# B&R Automation Studio project GAT (part 5)

#### FileOperations.st
```iecst
ACTION FileCopyOperation:

//	(* Export/Import recipes to/from USB *)
//    CASE hmiFile.Status.CopyStep OF
//        FILE_COPY_WAIT: (* Wait for export/import command *)
//            IF (hmiFile.Commands.ExportToUSB = TRUE) THEN
//                (* Check if USB device is available *)
//                IF (brsstrlen(ADR(MpFileManagerUIConnect.DeviceList.DeviceNames[1])) > 0) THEN
//
//                    (* USB is available proceed with export: select all files on the CF and trigger copy command *)
//                    IF (MpFileManagerUIConnect.DeviceList.SelectedIndex <> 0) THEN
//                        MpFileManagerUIConnect.DeviceList.SelectedIndex := 0;
//                        MpFileManagerUIConnect.File.MultiSelect := FALSE;
//                    ELSIF (MpFileManagerUIConnect.Status = mpFILE_UI_STATUS_IDLE) THEN
//
//                        IF NOT MpFileManagerUIConnect.File.MultiSelect THEN
//                            MpFileManagerUIConnect.File.MultiSelect := TRUE;
//                            FOR Index := 0 TO 49 DO
//                                MpFileManagerUIConnect.File.List.Items[Index].IsSelected := TRUE;
//                            END_FOR;
//                        ELSIF (brsstrlen(ADR(MpFileManagerUIConnect.File.List.Items[Index].Name)) = 0) THEN
//                            (* No files to copy, cancel operation *)
//                            hmiFile.Commands.ExportToUSB := FALSE;
//                        ELSE
//                            MpFileManagerUIConnect.File.Copy := TRUE;
//                            hmiFile.Status.CopyStep := FILE_COPY_TO_USB;
//                            hmiFile.Commands.ExportToUSB := FALSE;
//                        END_IF
//
//                    END_IF
//
//                ELSE
//                    (* No USB disk available, cancel operation *)
//                    hmiFile.Commands.ExportToUSB := FALSE;
//                END_IF
//
//            ELSIF hmiFile.Commands.ImportFromUSB THEN
//                (* Check if USB device is available *)
//                IF (brsstrlen(ADR(MpFileManagerUIConnect.DeviceList.DeviceNames[1])) > 0) THEN
//                    (* USB is available proceed with import: select all files on the USB and trigger copy command *)
//
//                    IF (MpFileManagerUIConnect.DeviceList.SelectedIndex <> 1) THEN
//                        MpFileManagerUIConnect.DeviceList.SelectedIndex := 1;
//                        MpFileManagerUIConnect.File.MultiSelect := FALSE;
//                    ELSIF MpFileManagerUIConnect.Status = mpFILE_UI_STATUS_IDLE THEN
//
//                        IF NOT MpFileManagerUIConnect.File.MultiSelect THEN
//                            MpFileManagerUIConnect.File.MultiSelect := TRUE;
//                            FOR Index := 0 TO ((SIZEOF(MpFileManagerUIConnect.File.List.Items)/SIZEOF(MpFileManagerUIConnect.File.List.Items[0])) - 1) DO
//                                MpFileManagerUIConnect.File.List.Items[Index].IsSelected := TRUE;
//                            END_FOR
//                        ELSIF (brsstrlen(ADR(MpFileManagerUIConnect.File.List.Items[Index].Name)) = 0) THEN
//                            (* No files to copy, cancel operation *)
//                            hmiFile.Commands.ImportFromUSB := FALSE;
//                        ELSE
//                            MpFileManagerUIConnect.File.Copy := TRUE;
//                            hmiFile.Status.CopyStep := FILE_COPY_FROM_USB;
//                            hmiFile.Commands.ImportFromUSB := FALSE;
//                        END_IF
//
//                    END_IF
//                ELSE
//                    (* No USB disk available, cancel operation *)
//                    hmiFile.Commands.ImportFromUSB := FALSE;
//                END_IF
//
//            END_IF
//
//        FILE_COPY_TO_USB: (* Navigate to USB device and paste files *)
//            IF (MpFileManagerUIConnect.Status = mpFILE_UI_STATUS_IDLE) THEN
//
//                IF (MpFileManagerUIConnect.DeviceList.SelectedIndex <> 1) THEN
//                    MpFileManagerUIConnect.DeviceList.SelectedIndex := 1;
//                    MpFileManagerUIConnect.File.MultiSelect := FALSE;
//                ELSE
//                    MpFileManagerUIConnect.File.Paste := TRUE;
//                END_IF
//
//            END_IF
//
//            IF MpFileManagerUIConnect.Status = mpFILE_UI_STATUS_PASTE THEN
//                hmiFile.Status.CopyStep := FILE_COPY_BUSY;
//            END_IF;
//
//        FILE_COPY_FROM_USB: (* Navigate to CF device and paste files *)
//            IF (MpFileManagerUIConnect.DeviceList.SelectedIndex <> 0) THEN
//                MpFileManagerUIConnect.DeviceList.SelectedIndex := 0;
//                MpFileManagerUIConnect.File.MultiSelect := FALSE;
//            ELSIF (MpFileManagerUIConnect.Status = mpFILE_UI_STATUS_IDLE) THEN
//                MpFileManagerUIConnect.File.Paste := TRUE;
//            END_IF
//
//            IF (MpFileManagerUIConnect.Status = mpFILE_UI_STATUS_PASTE) THEN
//                hmiFile.Status.CopyStep := FILE_COPY_BUSY;
//            END_IF
//
//        FILE_COPY_BUSY: (* Wait for copying done *)
//            IF (MpFileManagerUIConnect.MessageBox.Type = mpFILE_MSG_CONFIRM_OVERWRITE) OR (MpFileManagerUIConnect.MessageBox.Type = mpFILE_MSG_BUSY) THEN
//                (* TODO: Replace by confirm dialog *)
//                MpFileManagerUIConnect.MessageBox.Confirm := TRUE;
//            ELSIF MpFileManagerUIConnect.Status = mpFILE_UI_STATUS_IDLE THEN
//                hmiFile.Status.CopyStep := FILE_COPY_WAIT;
//            END_IF
//
//    END_CASE

END_ACTION
```

#### FIFOOperations.st - not listed in the package file held
```iecst
ACTION FIFOOperation:

	R_TRIG_CheckStatus(CLK := (MpFileManagerUIConnect.Status = mpFILE_UI_STATUS_CHANGE_DIR) OR
		(MpFileManagerUIConnect.Status = mpFILE_UI_STATUS_CHANGE_DEVICE) OR
		(MpFileManagerUIConnect.Status = mpFILE_UI_STATUS_CREATE));

	IF R_TRIG_CheckStatus.Q OR TON_ScanFolder.Q THEN
		HmiFile.Commands.CheckFolder := TRUE;
	END_IF

	// Autodelete oldest files based on scanning option
    CASE HmiFile.Status.DeleteStep OF

		FILE_DELETE_WAIT:
			// Wait for check the correct device selection
			TON_ScanFolder.IN := (HmiFile.Status.CurrentPage <> 'File_page');
			IF TON_ScanFolder.Q THEN
				TON_ScanFolder.IN := FALSE;
				HmiFile.Status.DeleteStep := FILE_SCAN_FOLDER_WAIT;
			END_IF

		FILE_SCAN_FOLDER_WAIT:
			// Wait for check for old files command
			IF (HmiFile.Commands.CheckFolder = TRUE) AND (MpFileManagerUIConnect.Status = mpFILE_UI_STATUS_IDLE) THEN
				HmiFile.Commands.CheckFolder := FALSE;
				HmiFile.Status.DeleteStep := FILE_SELECT_DEVICE;
				HmiFile.Parameters.OldSortOrder := MpFileManagerUIConnect.File.SortOrder;
			END_IF

		FILE_SELECT_DEVICE:
			// Sort by date so the oldest files are at the end
            IF (HmiFile.Status.DeviceName <> HmiFile.Parameters.Fifo.DeviceName) THEN
				FOR i := 0 TO ((SIZEOF(MpFileManagerUIConnect.DeviceList.DeviceNames)/SIZEOF(MpFileManagerUIConnect.DeviceList.DeviceNames[0])) - 1) DO
        			IF HmiFile.Parameters.Fifo.DeviceName = MpFileManagerUIConnect.DeviceList.DeviceNames[i] THEN
						MpFileManagerUIConnect.DeviceList.SelectedIndex := i;
					END_IF
    			END_FOR
            END_IF

            IF (HmiFile.Status.DeviceName = HmiFile.Parameters.Fifo.DeviceName) AND (MpFileManagerUIConnect.Status = mpFILE_UI_STATUS_IDLE) THEN
                HmiFile.Status.DeleteStep := FILE_SORT_BY_DATE;
            END_IF

		FILE_SORT_BY_DATE:
			// Sort by date so the oldest files are at the end
            IF (MpFileManagerUIConnect.File.SortOrder <> mpFILE_SORT_BY_MOD_TIME_DESC) THEN
                MpFileManagerUIConnect.File.SortOrder := mpFILE_SORT_BY_MOD_TIME_DESC;
            ELSIF (MpFileManagerUIConnect.Status = mpFILE_UI_STATUS_IDLE) THEN
                MpFileManagerUIConnect.File.Refresh := TRUE;
            END_IF

            IF (MpFileManagerUIConnect.Status = mpFILE_UI_STATUS_REFRESH) THEN
                HmiFile.Status.DeleteStep := FILE_CHECK_FOR_FILTER;
            END_IF

		FILE_CHECK_FOR_FILTER:
			// Check which delete filter is active
            IF (HmiFile.Parameters.Fifo.FifoType = FILE_FIFO_NUM_OF_FILES) THEN
                HmiFile.Status.DeleteStep := FILE_SELECT_OLDEST_FILES_0;
            ELSIF (HmiFile.Parameters.Fifo.FifoType = FILE_FIFO_SIZE_OF_FOLDER) THEN
				HmiFile.Status.DeleteStep := FILE_CALC_FOLDER_SIZE;
//			ELSIF (HmiFile.Parameters.Fifo.FifoType = FILE_FIFO_OLDER_THAN) THEN
//                HmiFile.Status.DeleteStep := FILE_SORT_BY_DATE;
			END_IF

		FILE_SELECT_OLDEST_FILES_0:
			// Scan and select all file over the filter setting
			IF (MpFileManagerUIConnect.Status = mpFILE_UI_STATUS_IDLE) THEN
				IF MpFileManagerUIConnect.File.PathInfo.FileCount > 1 THEN
           			MpFileManagerUIConnect.File.MultiSelect := TRUE;
				END_IF
				HmiFile.Status.AutoDeleteSelected := 0;
				FOR i := 0 TO ((SIZEOF(HmiFile.Status.FileNames)/SIZEOF(HmiFile.Status.FileNames[0])) - 1) DO
					IF i >= HmiFile.Parameters.Fifo.MaxNumberOfFiles THEN
						MpFileManagerUIConnect.File.List.Items[0].IsSelected := FALSE;
						IF (MpFileManagerUIConnect.File.List.Items[i].ItemType <> mpFILE_ITEM_TYPE_NONE) AND NOT MpFileManagerUIConnect.File.List.Items[i].IsFolder THEN
							MpFileManagerUIConnect.File.List.Items[i].IsSelected := TRUE;
							HmiFile.Status.AutoDeleteSelected := HmiFile.Status.AutoDeleteSelected + 1;
						END_IF
					END_IF
				END_FOR

				IF (HmiFile.Status.AutoDeleteSelected > 0) THEN
					HmiFile.Status.DeleteStep := FILE_DELETE_FILES;
				ELSE
					MpFileManagerUIConnect.File.MultiSelect := FALSE;
					HmiFile.Status.DeleteStep := FILE_RESET_SORT_BY;
				END_IF
			END_IF

		FILE_CALC_FOLDER_SIZE:
			// Calculate the overall file size in the open folder
				HmiFile.Status.FolderSize := 0;
				FOR i := 0 TO ((SIZEOF(HmiFile.Status.FileNames)/SIZEOF(HmiFile.Status.FileNames[0])) - 1) DO
					IF MpFileManagerUIConnect.File.List.Items[i].ItemType <> mpFILE_ITEM_TYPE_FOLDER THEN
						HmiFile.Status.FolderSize := HmiFile.Status.FolderSize + UDINT_TO_REAL(MpFileManagerUIConnect.File.List.Items[i].Size);
					END_IF
				END_FOR
				IF (HmiFile.Status.FolderSize > HmiFile.Parameters.Fifo.MaxFolderSize) THEN
					HmiFile.Status.DeleteStep := FILE_SELECT_OLDEST_FILES_1;
				ELSE
					HmiFile.Status.DeleteStep := FILE_RESET_SORT_BY;
				END_IF

		FILE_SELECT_OLDEST_FILES_1:
			// Scan and select all file over the filter setting
			IF (MpFileManagerUIConnect.Status = mpFILE_UI_STATUS_IDLE) THEN
				MpFileManagerUIConnect.File.List.Items[(MpFileManagerUIConnect.File.PathInfo.FileCount - 1)].IsSelected := TRUE;
				HmiFile.Status.DeleteStep := FILE_DELETE_FILES;
			END_IF

		FILE_DELETE_FILES:
			// Set command to delete the selected oldest files
			IF  (MpFileManagerUIConnect.Status = mpFILE_UI_STATUS_IDLE) THEN
				MpFileManagerUIConnect.File.Delete := TRUE;
			END_IF

			IF (MpFileManagerUIConnect.Status = mpFILE_UI_STATUS_DELETE) THEN
				HmiFile.Status.DeleteStep := FILE_CONFIRM_DELETE;
            END_IF

		FILE_CONFIRM_DELETE:
			// Confirm the file delete
            IF (MpFileManagerUIConnect.MessageBox.Type = mpFILE_MSG_CONFIRM_DELETE) THEN
                MpFileManagerUIConnect.MessageBox.Confirm := TRUE;
            ELSIF (MpFileManagerUIConnect.Status = mpFILE_UI_STATUS_IDLE) AND (MpFileManagerUIConnect.MessageBox.LayerStatus = 1) THEN
				IF (HmiFile.Parameters.Fifo.FifoType = FILE_FIFO_SIZE_OF_FOLDER) THEN
                	HmiFile.Status.DeleteStep := FILE_CALC_FOLDER_SIZE;
				ELSE
					HmiFile.Status.DeleteStep := FILE_RESET_SORT_BY;
					MpFileManagerUIConnect.File.MultiSelect := FALSE;
				END_IF
            END_IF

		FILE_RESET_SORT_BY:
			// Restore old sort order
            IF (MpFileManagerUIConnect.File.SortOrder <> HmiFile.Parameters.OldSortOrder) THEN
                MpFileManagerUIConnect.File.SortOrder := HmiFile.Parameters.OldSortOrder;
            ELSIF (MpFileManagerUIConnect.Status = mpFILE_UI_STATUS_IDLE) THEN
                MpFileManagerUIConnect.File.Refresh := TRUE;
            END_IF

            IF (MpFileManagerUIConnect.Status = mpFILE_UI_STATUS_REFRESH) THEN
                HmiFile.Status.DeleteStep := FILE_DELETE_WAIT;
				IF (MpFileManagerUIConnect.MessageBox.Type = mpFILE_MSG_BUSY) THEN
					MpFileManagerUIConnect.MessageBox.Confirm := TRUE;
				END_IF
            END_IF
	END_CASE

	TON_ScanFolder(PT := DINT_TO_TIME(HmiFile.Parameters.Fifo.ScanInterval * 60000));

END_ACTION
```

### Package Logical/Infrastructure/Usb - Package for USB handling for mapp Framework

### Program Logical/Infrastructure/Usb/UsbMgr (IEC) - Usb manager

#### UsbMgr.st - Init, cyclic, exit code
```iecst
//*********************************************************************************
// Copyright: B&R Industrial Automation GmbH
// Author: B&R Industrial Automation GmbH
// Created: April 12, 2022
// Description: This task automatically detects and (un)links USB storage devices
//*********************************************************************************

PROGRAM _INIT

	DevLinkCtrl.FUB.DevLink_0.enable := FALSE;
	DevLinkCtrl.FUB.DevUnlink_0.enable := FALSE;
	DevLinkCtrl.FUB.UsbNodeGet_0.enable := FALSE;
	DevLinkCtrl.FUB.UsbNodeListGet_0.enable := FALSE;
	DevLinkCtrl.FUB.DevLink_0();
	DevLinkCtrl.FUB.DevUnlink_0();
	DevLinkCtrl.FUB.UsbNodeGet_0();
	DevLinkCtrl.FUB.UsbNodeListGet_0();

	FOR i := 0 TO MAX_IDX_USB_DEV_LIST DO
		AttachedUSB[i] := FALSE;
		gUSBAvailable[i] := FALSE;
	END_FOR

END_PROGRAM

PROGRAM _CYCLIC

	CASE DevLinkCtrl.Step OF
		STATE_WAIT:
			// Update USB info list if the node list has changed
			IF (brsmemcmp(ADR(DevLinkCtrl.Parameters.NodeList), ADR(LastNodeList), SIZEOF(LastNodeList)) <> 0) THEN
				DevLinkCtrl.Commands.GetUSBInfo := TRUE;
				// Preserve the previously created drive information in case the order has changed when unplugging a device
				FOR DevLinkCtrl.Parameters.Index := 0 TO MAX_IDX_USB_DEV_LIST DO
					FOR i := 0 TO MAX_IDX_USB_DEV_LIST DO
						IF ((DevLinkCtrl.Parameters.NodeList[DevLinkCtrl.Parameters.Index] = LastNodeList[i]) AND
							(DevLinkCtrl.Parameters.Index <> i) AND (LastNodeList[i] <> 0)) THEN
							brsmemcpy(ADR(TempUSBInfo), ADR(DevLinkCtrl.Parameters.NodeInfoList[DevLinkCtrl.Parameters.Index]), SIZEOF(TempUSBInfo));
							brsmemcpy(ADR(DevLinkCtrl.Parameters.NodeInfoList[DevLinkCtrl.Parameters.Index]), ADR(DevLinkCtrl.Parameters.NodeInfoList[i]), SIZEOF(TempUSBInfo));
							brsmemcpy(ADR(DevLinkCtrl.Parameters.NodeInfoList[i]), ADR(TempUSBInfo), SIZEOF(TempUSBInfo));
							brsmemcpy(ADR(TempFileDeviceName), ADR(DevLinkCtrl.Parameters.FileDevName[DevLinkCtrl.Parameters.Index]), SIZEOF(TempFileDeviceName));
							brsmemcpy(ADR(DevLinkCtrl.Parameters.FileDevName[DevLinkCtrl.Parameters.Index]), ADR(DevLinkCtrl.Parameters.FileDevName[i]), SIZEOF(TempFileDeviceName));
							brsmemcpy(ADR(DevLinkCtrl.Parameters.FileDevName[i]), ADR(TempFileDeviceName), SIZEOF(TempFileDeviceName));
							TempFileDeviceHandle := DevLinkCtrl.Parameters.FileDevHandle[DevLinkCtrl.Parameters.Index];
							DevLinkCtrl.Parameters.FileDevHandle[DevLinkCtrl.Parameters.Index] := DevLinkCtrl.Parameters.FileDevHandle[i];
							DevLinkCtrl.Parameters.FileDevHandle[i] := TempFileDeviceHandle;
						END_IF
					END_FOR
				END_FOR
				brsmemcpy(ADR(LastNodeList), ADR(DevLinkCtrl.Parameters.NodeList), SIZEOF(LastNodeList));
			END_IF

			FOR DevLinkCtrl.Parameters.Index := 0 TO MAX_IDX_USB_DEV_LIST DO
				// Skip if loading USB list information
				IF DevLinkCtrl.Commands.GetUSBInfo THEN
					EXIT;
				END_IF
				// Always keep devices linked when available
				IF ((DevLinkCtrl.Parameters.FileDevHandle[DevLinkCtrl.Parameters.Index] = 0) AND AttachedUSB[DevLinkCtrl.Parameters.Index]
					AND (DevLinkCtrl.Parameters.NodeList[DevLinkCtrl.Parameters.Index] <> 0)) THEN
					DevLinkCtrl.Commands.DevLink := TRUE;
					EXIT;
				END_IF
				// Unlink device if it is not connected anymore
				IF ((DevLinkCtrl.Parameters.FileDevHandle[DevLinkCtrl.Parameters.Index] <> 0) AND
					(DevLinkCtrl.Parameters.NodeInfoList[DevLinkCtrl.Parameters.Index].interfaceClass <> 8)) THEN
					DevLinkCtrl.Commands.DevUnlink := TRUE;
					EXIT;
				END_IF
			END_FOR

			// Check for USB devices every 3 seconds
			TON_0.PT := t#3s;
			IF (TON_0.Q AND NOT DevLinkCtrl.Commands.GetUSBInfo AND NOT DevLinkCtrl.Commands.DevLink AND NOT DevLinkCtrl.Commands.DevUnlink) THEN
				DevLinkCtrl.Commands.GetUSBList := TRUE;
				TON_0.IN := FALSE;
			ELSE
				TON_0.IN := TRUE;
			END_IF
			TON_0();

			IF DevLinkCtrl.Commands.GetUSBInfo THEN
				// Get USB info Commands
				DevLinkCtrl.Commands.GetUSBInfo := FALSE;
				brsmemset(ADR(DevLinkCtrl.Parameters.NodeInfoList), 0, SIZEOF(DevLinkCtrl.Parameters.NodeInfoList));
				DevLinkCtrl.Step := STATE_GET_USB_INFO;
				DevLinkCtrl.Parameters.Index := 0;
			ELSIF DevLinkCtrl.Commands.GetUSBList THEN
				// Get USB list Commands
				DevLinkCtrl.Commands.GetUSBList := FALSE;
				brsmemset(ADR(DevLinkCtrl.Parameters.NodeList), 0, SIZEOF(DevLinkCtrl.Parameters.NodeList));
				DevLinkCtrl.Step := STATE_GET_USB_LIST;
			ELSIF DevLinkCtrl.Commands.DevLink THEN
				// Link Commands
				DevLinkCtrl.Commands.DevLink := FALSE;
				DevLinkCtrl.Step := STATE_DEV_LINK;
			ELSIF DevLinkCtrl.Commands.DevUnlink THEN
				// Unlink Commands
				DevLinkCtrl.Commands.DevUnlink := FALSE;
				DevLinkCtrl.Step := STATE_DEV_UNLINK;
			END_IF

		STATE_GET_USB_LIST:
			// Set FUB parameters
			DevLinkCtrl.FUB.UsbNodeListGet_0.enable := TRUE;
			DevLinkCtrl.FUB.UsbNodeListGet_0.bufferSize := SIZEOF(DevLinkCtrl.Parameters.NodeList);
			DevLinkCtrl.FUB.UsbNodeListGet_0.pBuffer := ADR(DevLinkCtrl.Parameters.NodeList);

			// Error handling
			IF ((DevLinkCtrl.FUB.UsbNodeListGet_0.status = ERR_OK) OR (DevLinkCtrl.FUB.UsbNodeListGet_0.status = asusbERR_USB_NOTFOUND)) THEN
				DevLinkCtrl.Step := STATE_WAIT;
				DevLinkCtrl.FUB.UsbNodeListGet_0.enable := FALSE;
			ELSIF ((DevLinkCtrl.FUB.UsbNodeListGet_0.status <> ERR_FUB_BUSY) AND (DevLinkCtrl.FUB.UsbNodeListGet_0.status <> ERR_FUB_ENABLE_FALSE)
				AND (DevLinkCtrl.FUB.UsbNodeListGet_0.status <> asusbERR_USB_NOTFOUND)) THEN
				DevLinkCtrl.Step := STATE_ERROR_USB;
				DevLinkCtrl.Parameters.ErrorID := DevLinkCtrl.FUB.UsbNodeListGet_0.status;
				DevLinkCtrl.FUB.UsbNodeListGet_0.enable := FALSE;
			END_IF

			DevLinkCtrl.FUB.UsbNodeListGet_0();

		STATE_GET_USB_INFO:
			// Set FUB parameters
			DevLinkCtrl.FUB.UsbNodeGet_0.bufferSize := SIZEOF(DevLinkCtrl.Parameters.NodeInfoList[DevLinkCtrl.Parameters.Index]);
			DevLinkCtrl.FUB.UsbNodeGet_0.enable := TRUE;
			DevLinkCtrl.FUB.UsbNodeGet_0.nodeId := DevLinkCtrl.Parameters.NodeList[DevLinkCtrl.Parameters.Index];
			DevLinkCtrl.FUB.UsbNodeGet_0.pBuffer := ADR(DevLinkCtrl.Parameters.NodeInfoList[DevLinkCtrl.Parameters.Index]);

			// Check if DevLinkCtrl.Parameters.Index contains an entry
			IF (DevLinkCtrl.Parameters.NodeList[DevLinkCtrl.Parameters.Index] = 0) THEN
				DevLinkCtrl.FUB.UsbNodeGet_0.enable := TRUE;
				brsmemset(ADR(DevLinkCtrl.Parameters.NodeInfoList[DevLinkCtrl.Parameters.Index]), 0, SIZEOF(DevLinkCtrl.Parameters.NodeInfoList[DevLinkCtrl.Parameters.Index]));
				DevLinkCtrl.Parameters.Index := DevLinkCtrl.Parameters.Index + 1;
			END_IF

			// Error handling
			IF (DevLinkCtrl.FUB.UsbNodeGet_0.status = ERR_OK) THEN
				DevLinkCtrl.FUB.UsbNodeGet_0.enable := FALSE;
				DevLinkCtrl.Parameters.Index := DevLinkCtrl.Parameters.Index + 1;
			ELSIF ((DevLinkCtrl.FUB.UsbNodeGet_0.status <> ERR_FUB_BUSY) AND (DevLinkCtrl.FUB.UsbNodeGet_0.status <> ERR_FUB_ENABLE_FALSE)) THEN
				DevLinkCtrl.Step := STATE_ERROR_USB;
				DevLinkCtrl.Parameters.ErrorID := DevLinkCtrl.FUB.UsbNodeGet_0.status;
				DevLinkCtrl.FUB.UsbNodeGet_0.enable := FALSE;
			END_IF

			// End of list reached
			IF (DevLinkCtrl.Parameters.Index > MAX_IDX_USB_DEV_LIST) THEN
				DevLinkCtrl.FUB.UsbNodeGet_0.enable := FALSE;
				DevLinkCtrl.Step := STATE_WAIT;
				FOR DevLinkCtrl.Parameters.Index := 0 TO MAX_IDX_USB_DEV_LIST DO
					IF (DevLinkCtrl.Parameters.NodeInfoList[DevLinkCtrl.Parameters.Index].interfaceClass = 8) THEN
						AttachedUSB[DevLinkCtrl.Parameters.Index] := TRUE;
					ELSE
						AttachedUSB[DevLinkCtrl.Parameters.Index] := FALSE;
						gUSBAvailable[DevLinkCtrl.Parameters.Index] := FALSE;
					END_IF
				END_FOR
			END_IF

			DevLinkCtrl.FUB.UsbNodeGet_0();

		STATE_DEV_LINK:
            // Set FUB parameters
			DevLinkCtrl.FUB.DevLink_0.enable := TRUE;
			DevLinkCtrl.FUB.DevLink_0.pDevice := ADR(DevLinkCtrl.Parameters.FileDevName[DevLinkCtrl.Parameters.Index]);
			DevLinkCtrl.Parameters.LinkParam := '/DEVICE=';
			brsstrcat(ADR(DevLinkCtrl.Parameters.LinkParam), ADR(DevLinkCtrl.Parameters.NodeInfoList[DevLinkCtrl.Parameters.Index].ifName));
			DevLinkCtrl.FUB.DevLink_0.pParam := ADR(DevLinkCtrl.Parameters.LinkParam);

			// Error handling
			IF (DevLinkCtrl.FUB.DevLink_0.status = ERR_OK) THEN
				DevLinkCtrl.Parameters.FileDevHandle[DevLinkCtrl.Parameters.Index] := DevLinkCtrl.FUB.DevLink_0.handle;
				DevLinkCtrl.Step := STATE_WAIT;
				DevLinkCtrl.FUB.DevLink_0.enable := FALSE;
				FOR i := 0 TO MAX_IDX_USB_DEV_LIST DO
					gUSBAvailable[i] := AttachedUSB[i];
				END_FOR
			ELSIF ((DevLinkCtrl.FUB.DevLink_0.status <> ERR_FUB_BUSY) AND (DevLinkCtrl.FUB.DevLink_0.status <> ERR_FUB_ENABLE_FALSE)) THEN
				DevLinkCtrl.Step := STATE_ERROR_USB;
				DevLinkCtrl.Parameters.ErrorID := DevLinkCtrl.FUB.DevLink_0.status;
				DevLinkCtrl.FUB.DevLink_0.enable := FALSE;
			END_IF

			DevLinkCtrl.FUB.DevLink_0();

		STATE_DEV_UNLINK:
			// Set FUB parameters
			DevLinkCtrl.FUB.DevUnlink_0.enable := TRUE;
			DevLinkCtrl.FUB.DevUnlink_0.handle := DevLinkCtrl.Parameters.FileDevHandle[DevLinkCtrl.Parameters.Index];

			// Check if we have a handle
			IF (DevLinkCtrl.Parameters.FileDevHandle[DevLinkCtrl.Parameters.Index] = 0) THEN
				DevLinkCtrl.FUB.DevUnlink_0.enable := FALSE;
				DevLinkCtrl.Step := STATE_WAIT;
			END_IF

			// Error handling
			IF (DevLinkCtrl.FUB.DevUnlink_0.status = ERR_OK) THEN
				DevLinkCtrl.Parameters.FileDevHandle[DevLinkCtrl.Parameters.Index] := 0;
				DevLinkCtrl.FUB.DevUnlink_0.enable := FALSE;
				DevLinkCtrl.Step := STATE_WAIT;
			ELSIF ((DevLinkCtrl.FUB.DevUnlink_0.status <> ERR_FUB_BUSY) AND (DevLinkCtrl.FUB.DevUnlink_0.status <> ERR_FUB_ENABLE_FALSE)) THEN
				DevLinkCtrl.Step := STATE_ERROR_USB;
				DevLinkCtrl.Parameters.ErrorID := DevLinkCtrl.FUB.DevUnlink_0.status;
				DevLinkCtrl.FUB.DevUnlink_0.enable := FALSE;
			END_IF

			DevLinkCtrl.FUB.DevUnlink_0();

		STATE_ERROR_USB:
			// Delete error ID and go back to wait step when error is acknowledged
			IF DevLinkCtrl.Commands.ErrAck THEN
				DevLinkCtrl.Parameters.ErrorID := 0;
				DevLinkCtrl.Commands.ErrAck := FALSE;
				DevLinkCtrl.Step := STATE_WAIT;
			END_IF

	END_CASE;

END_PROGRAM

PROGRAM _EXIT

	// Insert code here

END_PROGRAM
```

#### UsbMgr.typ - Local data types
```iecst
(*********************************************************************************
 * Copyright: Bernecker + Rainer
 * Author:    MITC
 * Created:   21 October, 2015/1:30 PM
 *********************************************************************************
 * DevLinkTask data types of project
 *********************************************************************************)

TYPE
	StepType :
		( (*enumeration of the possible machine states*)
		STATE_WAIT := 0, (*waiting for cmds*)
		STATE_GET_USB_LIST, (*getting list of usb devices*)
		STATE_GET_USB_INFO, (*getting info from a usb device*)
		STATE_DEV_LINK, (*linking device*)
		STATE_DEV_UNLINK, (*unlinking device*)
		STATE_ERROR_USB (*some FUB returned an error*)
		);
	CommandType : 	STRUCT  (*possible machine cmds*)
		GetUSBList : BOOL; (*get usb list cmd*)
		GetUSBInfo : BOOL; (*get usb info cmd*)
		DevLink : BOOL; (*link cmd*)
		DevUnlink : BOOL; (*unlink cmd*)
		ErrAck : BOOL; (*error acknowledge cmd*)
	END_STRUCT;
	DevLink_FUBType : 	STRUCT  (*contains all needed FileIO FUBs*)
		UsbNodeListGet_0 : UsbNodeListGet;
		UsbNodeGet_0 : UsbNodeGet;
		UsbMsDeviceReady_0 : UsbMsDeviceReady;
		DevLink_0 : DevLink;
		DevUnlink_0 : DevUnlink;
	END_STRUCT;
	DevLinkCtrlType : 	STRUCT  (*Control structure which contains everything necessary for the file handling machine*)
		Step : StepType; (*actual step*)
		Cmd : CommandType; (*when in STATE_WAIT a cmd with value true will change the machine state*)
		FUB : DevLink_FUBType; (*all DevLink FUBs*)
		Params : ParamsType; (*parameters like file device, error ID, Buffer, ...*)
	END_STRUCT;
	ParamsType : 	STRUCT  (*Parameter structure*)
		ErrorID : UINT; (*the error id from a FUB is stored here in case of error*)
		NodeList : ARRAY[0..MAX_IDX_USB_DEV_LIST]OF UDINT; (*List of connected usb devices*)
		NodeInfoList : ARRAY[0..MAX_IDX_USB_DEV_LIST]OF usbNode_typ; (*Buffer for usb info*)
		FileDevName : ARRAY[0..MAX_IDX_USB_DEV_LIST]OF STRING[30]; (*file device names*)
		FileDevHandle : ARRAY[0..MAX_IDX_USB_DEV_LIST]OF UDINT; (*needed for unlinking the device again*)
		LinkParam : STRING[30]; (*param string to link a device*)
		Index : USINT; (*list index*)
	END_STRUCT;
END_TYPE
```

#### UsbMgr.var - Local variables
```iecst
(*Function Blocks*)
VAR
	TON_0 : TON; (*Tiimer to refresh available usb devices*)
END_VAR
(*Structure Types*)
VAR
	DevLinkCtrl : DevLinkControlType := (0); (*DevLink control structure*)
	TempUSBInfo : usbNode_typ := (0); (*Temporary info structure*)
END_VAR
(*Variables*)
VAR
	LastNodeList : ARRAY[0..MAX_IDX_USB_DEV_LIST] OF UDINT; (*Temporary variable to check if the node list has changed*)
	AttachedUSB : ARRAY[0..MAX_IDX_USB_DEV_LIST] OF BOOL := [2(FALSE)]; (*Flags for whether the USB devices are detected*)
	TempFileDeviceName : STRING[30] := ''; (*Temporary file device name*)
	TempFileDeviceHandle : UDINT := 0; (*Temporary file device handle*)
	i : USINT := 0; (*index to loop through ussb devices*)
	tempDigit : STRING[80];
END_VAR
```

### Package Logical/Infrastructure/Report - Package for mapp Report Framework

### Program Logical/Infrastructure/Report/ReportMgr (IEC) - Report manager

#### ReportMgt.var
```iecst
(********************************************************************
 * COPYRIGHT -- Bernecker + Rainer
 ********************************************************************
 * Program: FolderHandling
 * File: FolderHandling.var
 * Author: Bernecker + Rainer
 * Created: December , 2020
 ********************************************************************
 * Local variables of program Alarm Management
 ********************************************************************)
(*Function Block Declaration*)
VAR
	MpFileManagerUIConnect : MpFileManagerUIConnectType := (DeviceList:=(DeviceNames:=['mappReportFiles',9('')]));
	MpFileManagerUI_0 : MpFileManagerUI;
	TON_0 : TON := (0); (*Timer to wait before refresh*)
	MpReportCore_0 : MpReportCore := (0); (*Core variable for MpReport*)
	LanguageSelect_0 : LanguageSelect := (LanguageSelection:=['en','de'],SelectedIndex:=0);
	DirCreate_0 : DirCreate;
END_VAR
(*Report Management Variables*)
VAR
	EnableDelete : BOOL := TRUE; (*HMI control bit*)
	EnableGenerate : BOOL := TRUE; (*HMI control bit*)
	Refresh : BOOL := 0; (*strrt refresh process*)
	StartGenerate : BOOL := 0; (*variable for interaction with Visualization*)
	DeleteReport : BOOL := 0; (*Start deleting a Report*)
	i : USINT := 0; (*index for save filenames in a array*)
	DisplayFileNameIndex : USINT := 0; (*index of selected file for display in table in mappView*)
	DisplayFileName : ARRAY[0..49] OF STRING[255] := [50('')]; (*Displayed Files for mappView*)
	SetLanguage : STRING[80] := ''; (*Set the current language*)
	TableConfig : STRING[80];
	StrSelectedFile : STRING[256] := '0'; (*Gives the path of selected report to pdfViewer in mappView*)
END_VAR
(*Constants*)
VAR CONSTANT
	REPORT_DEVICE : STRING[80] := 'mappReportFiles'; (*Constant contains filedevice for save reports *)
	REPORT_NAME : STRING[80] := 'Report'; (*Constant contains name of Report*)
	STR_FILE_DEVICE : STRING[80] := '/FileDevice:mappReport/'; (*File Device*)
	LOCAL_FOLDER : STRING[10] := 'Report';
END_VAR
```

#### ReportMgt.st
```iecst
//*********************************************************************************
//* Copyright: B&R Industrial Automation GmbH
//* Author:    B&R Industrial Automation GmbH
//* Created:   30. Sep 2020/08:00
//* Description: Tasks FOR report control. The Report Control handling is done in this task.
//********************************************************************************

PROGRAM _INIT

	// Create folder for this component on the user file device
	DirCreate_0(enable := TRUE, pDevice := ADR('UserPartition'), pName := ADR(LOCAL_FOLDER));

	// Check if folder already exist and if so disabled the function block call
	IF DirCreate_0.status = fiERR_DIR_ALREADY_EXIST THEN
		DirCreate_0(enable := FALSE);
	END_IF

	// Init mapp function blocks
	MpReportCore_0.Enable := TRUE;
	MpReportCore_0.MpLink := ADR(gMpLinkReport);
	MpReportCore_0.Name := ADR(REPORT_NAME);
	MpReportCore_0.DeviceName := ADR(REPORT_DEVICE);
	MpFileManagerUI_0.MpLink := ADR(gMpLinkFileManagerUIReport);
	MpFileManagerUI_0.UIConnect := ADR(MpFileManagerUIConnect);
	MpFileManagerUI_0.Enable := TRUE;
	// Filter for pdf files
	MpFileManagerUIConnect.File.Filter := '*.pdf';
END_PROGRAM

PROGRAM _CYCLIC
	// Configure visible file list
	brsstrcpy(ADR(TableConfig), ADR('{ "specRows": [{"from":'));
	brsitoa(MpFileManagerUIConnect.File.PathInfo.FileCount, ADR(TableConfig) + brsstrlen(ADR(TableConfig)));
	brsstrcat(ADR(TableConfig),  ADR(',"to":49, "visible":false}]}'));

	// Refresh report action
	RefreshReport;

	// Reset ErrorReset command
	IF NOT MpReportCore_0.Error THEN
		MpReportCore_0.ErrorReset := FALSE;
	END_IF

	// Function block calls
	MpReportCore_0();
	MpFileManagerUI_0();
END_PROGRAM

PROGRAM _EXIT
	// Disable and call mapp function blocks
	MpReportCore_0.Enable := FALSE;
	MpFileManagerUI_0.Enable := FALSE;
	MpReportCore_0();
	MpFileManagerUI_0();
END_PROGRAM
```

### Program Logical/Infrastructure/Report/ReportMgt (IEC)

#### ReportMgt.st - Cyclic code
```iecst
//*********************************************************************************
//* Copyright: B&R Industrial Automation GmbH
//* Author:    B&R Industrial Automation GmbH
//* Created:   30. Sep 2020/08:00
//* Description: Tasks FOR report control. The Report Control handling is done in this task.
//********************************************************************************

PROGRAM _INIT

	//Create folder for this component on the user file device
	DirCreate_New(enable := TRUE, pDevice := ADR('userPartition'), pName := ADR(LOCAL_FOLDER));

	//Check if folder already exist and if so disabled the function block call
	IF DirCreate_New.status = fiERR_DIR_ALREADY_EXIST THEN
		DirCreate_New(enable := FALSE);
	END_IF

	// Init mapp function blocks
	MpReportCore_0.Enable := TRUE;
	MpReportCore_0.MpLink := ADR(gMpLinkReport);
	MpReportCore_0.Name := ADR(REPORT_NAME);
	MpReportCore_0.DeviceName := ADR(REPORT_DEVICE);
	MpFileManagerUI_0.MpLink := ADR(gMpLinkFileManagerUIReport);
	MpFileManagerUI_0.UIConnect := ADR(MpFileManagerUIConnect);
	MpFileManagerUI_0.Enable := TRUE;
	// Filter for pdf files
	MpFileManagerUIConnect.File.Filter := '*.pdf';
END_PROGRAM

PROGRAM _CYCLIC
	// Configure visible file list
	brsstrcpy(ADR(TableConfig), ADR('{ "specRows": [{"from":'));
	brsitoa(MpFileManagerUIConnect.File.PathInfo.FileCount, ADR(TableConfig) + brsstrlen(ADR(TableConfig)));
	brsstrcat(ADR(TableConfig),  ADR(',"to":49, "visible":false}]}'));

	// Refresh report action
	RefreshReport;

	// Reset ErrorReset command
	IF NOT MpReportCore_0.Error THEN
		MpReportCore_0.ErrorReset := FALSE;
	END_IF

	// Function block calls
	MpReportCore_0();
	MpFileManagerUI_0();
END_PROGRAM

PROGRAM _EXIT
	// Disable and call mapp function blocks
	MpReportCore_0.Enable := FALSE;
	MpFileManagerUI_0.Enable := FALSE;
	MpReportCore_0();
	MpFileManagerUI_0();
END_PROGRAM
```

#### ReportMgt.typ - Local data types
```iecst
TYPE
	LanguageSelect : 	STRUCT
		LanguageSelection : ARRAY[0..1]OF STRING[80] := ['en','de'];
		SelectedIndex : INT := 0;
	END_STRUCT;
END_TYPE
```

#### ReportMgt.var - Local variables
```iecst
(********************************************************************
 * COPYRIGHT -- Bernecker + Rainer
 ********************************************************************
 * Program: FolderHandling
 * File: FolderHandling.var
 * Author: Bernecker + Rainer
 * Created: December , 2020
 ********************************************************************
 * Local variables of program Alarm Management
 ********************************************************************)
(*Function Block Declaration*)
VAR
	MpFileManagerUIConnect : MpFileManagerUIConnectType := (DeviceList:=(DeviceNames:=['mappReport',9('')]));
	MpFileManagerUI_0 : MpFileManagerUI;
	TON_0 : TON := (0); (*Timer to wait before refresh*)
	MpReportCore_0 : MpReportCore := (0); (*Core variable for MpReport*)
	LanguageSelect_0 : LanguageSelect := (LanguageSelection:=['en','de'],SelectedIndex:=0);
	DirCreate_New : DirCreate;
END_VAR
(*Report Management Variables*)
VAR
	EnableDelete : BOOL := TRUE; (*HMI control bit*)
	EnableGenerate : BOOL := TRUE; (*HMI control bit*)
	Refresh : BOOL := 0; (*strrt refresh process*)
	StartGenerate : BOOL := 0; (*variable for interaction with Visualization*)
	DeleteReport : BOOL := 0; (*Start deleting a Report*)
	i : USINT := 0; (*index for save filenames in a array*)
	DisplayFileNameIndex : USINT := 0; (*index of selected file for display in table in mappView*)
	DisplayFileName : ARRAY[0..49] OF STRING[255] := [50('')]; (*Displayed Files for mappView*)
	SetLanguage : STRING[80] := ''; (*Set the current language*)
	TableConfig : STRING[80];
	StrSelectedFile : STRING[256] := '0'; (*Gives the path of selected report to pdfViewer in mappView*)
END_VAR
(*Constants*)
VAR CONSTANT
	REPORT_DEVICE : STRING[80] := 'mappReport'; (*Constant contains filedevice for save reports *)
	REPORT_NAME : STRING[80] := 'Report'; (*Constant contains name of Report*)
	STR_FILE_DEVICE : STRING[80] := '/FileDevice:mappReport/'; (*File Device*)
	LOCAL_FOLDER : STRING[10] := 'Report';
END_VAR
```

#### RefreshReport.st - Showing Report in list
```iecst
ACTION RefreshReport:

    // Generate process
	IF StartGenerate = TRUE THEN
		MpReportCore_0.Language := ADR(LanguageSelect_0.LanguageSelection[LanguageSelect_0.SelectedIndex]);
		MpReportCore_0.Generate := TRUE;

		IF MpReportCore_0.CommandDone = TRUE THEN

			StartGenerate := FALSE;
			Refresh := TRUE;
			EnableGenerate := FALSE;
		END_IF

	ELSE
		MpReportCore_0.Generate := FALSE;
	END_IF

    // Deleting process
	IF DeleteReport = TRUE THEN
		MpFileManagerUIConnect.File.Delete := TRUE;
		MpFileManagerUIConnect.MessageBox.Confirm := TRUE;
		DeleteReport := FALSE;
		Refresh := TRUE;
		EnableDelete := FALSE;
    END_IF

	// Refresh process
	IF Refresh = TRUE THEN
		TON_0(IN := TRUE, PT := T#2s);
		IF TON_0.Q = TRUE THEN
			Refresh := FALSE;
			TON_0(IN := FALSE, PT := T#2s);
			MpFileManagerUIConnect.File.Refresh := TRUE;
		END_IF
	END_IF

    // reset enable attribute for buttons
	IF Refresh = FALSE THEN
		EnableDelete := TRUE;
		EnableGenerate := TRUE;
	END_IF

    // Save Filenames to a seperate array for display in Table
	FOR i := 0 TO 49 DO
        DisplayFileName[i] := MpFileManagerUIConnect.File.List.Items[i].Name;
        // if selected set a index for display selected file in table
		IF DisplayFileNameIndex = i THEN
			MpFileManagerUIConnect.File.List.Items[i].IsSelected := TRUE;
		END_IF
	END_FOR

    // String for pdfViewer to display right report
	StrSelectedFile := CONCAT(STR_FILE_DEVICE, MpFileManagerUIConnect.File.List.Items[DisplayFileNameIndex].Name);

	IF LanguageSelect_0.SelectedIndex = 0 THEN
		SetLanguage := 'en';
	ELSE
		SetLanguage := 'de';
	END_IF

END_ACTION
```

### Package Logical/Infrastructure/Recipe - Package for mapp Recipe Framework

### Program Logical/Infrastructure/Recipe/RecipeMgr (IEC) - Recipe manager

#### RecipeMgr.st - Init, cyclic, exit code
```iecst
//***********************************************************************
// Copyright: B&R Industrial Automation GmbH
// Author: B&R Industrial Automation GmbH
// Created: Jan 1, 2022
// Description: Tasks for recipe control.
//***********************************************************************

PROGRAM _INIT

	// Create folder for this component on the user file device
	DirCreate_0(enable := TRUE, pDevice := ADR('UserPartition'), pName := ADR(LOCAL_FOLDER));

	// Check if folder already exist and if so disabled the function block call
	IF DirCreate_0.status = fiERR_DIR_ALREADY_EXIST THEN
		DirCreate_0(enable := FALSE);
	END_IF

	// Initialize mapp function blocks
	// By default, the Framework sets up an XML recipe system. To swtich to the CSV format, refer to the "Change Recipe Format"
	// page in the AS Help (GUID 2052b3a5-f59b-45f9-9fcd-3289c93401af)
	MpRecipeUISetup.Confirmation.RecipeDelete := TRUE;
	MpRecipeUISetup.RecipeListSize := 10;
	MpRecipeUISetup.RecipeListScrollWindow := 0;
	MpRecipeUISetup.AutoLoadHeader := TRUE;
	MpRecipeUIConnect.New.FileName := 'newRecipe.par';
	MpRecipeUIConnect.Recipe.Filter := '*par';
	MpRecipeUI_0.MpLink := ADR(gMpLinkRecipeXml);
	MpRecipeUI_0.Enable := TRUE;
	MpRecipeUI_0.UIConnect := ADR(MpRecipeUIConnect);
	MpRecipeUI_0.UISetup := MpRecipeUISetup;
	MpRecipeUI_0();

	HmiRecipe.Parameters.Category := PARAMETERS_CATEGORY;
	HmiRecipe.Parameters.DeviceDataProvider[0] := '{"value":"mappRecipeFiles","text":"CF/PLC"}';
	HmiRecipe.Parameters.DeviceName := 'mappRecipeFiles';
	MpRecipe_0.MpLink := ADR(gMpLinkRecipeXml);
	MpRecipe_0.Enable := TRUE;
	MpRecipe_0.Category := ADR(HmiRecipe.Parameters.Category);
	MpRecipe_0.DeviceName := ADR(HmiRecipe.Parameters.DeviceName);
    MpRecipe_0.FileName := ADR(HmiRecipe.Parameters.FileName);
	MpRecipe_0.Header := ADR(Header);

	// Wait for MpRecipe_0 to activate. This must be active before you can call the RegPar function blocks, which is below.
	WHILE NOT(MpRecipe_0.Active OR MpRecipe_0.Error) DO
		MpRecipe_0();
	END_WHILE

	// Register the preview variables to the recipe. These preview variables are a buffer between the recipe system and the
	// variables used at runtime on the machine (Parameters, MachineSettings). By using these preview variables, you can
	// preview and edit a recipe on the HMI without actually loading it to the machine. For more details, refer to the
	// "Recipe System Design" page in the AS Help (GUID 3ccd7409-0b52-4bbc-a93a-4010f6db414c).

    MpRecipeRegPar_PreviewPar.MpLink := ADR(gMpLinkRecipeXml);
	MpRecipeRegPar_PreviewPar.Enable := TRUE;
	MpRecipeRegPar_PreviewPar.PVName := ADR('RecipeMgr:ParametersPreview');
	MpRecipeRegPar_PreviewPar.Category := ADR(PARAMETERS_CATEGORY);
	MpRecipeRegPar_PreviewPar();

	MpRecipeRegPar_PreviewCfg.MpLink := ADR(gMpLinkRecipeXml);
	MpRecipeRegPar_PreviewCfg.Enable := TRUE;
	MpRecipeRegPar_PreviewCfg.PVName := ADR('RecipeMgr:MachineSettingsPreview');
	MpRecipeRegPar_PreviewCfg.Category := ADR(MACHINE_CONFIGURATION_CATEGORY);
	MpRecipeRegPar_PreviewCfg();

	// Wait for RegPar function blocks to activate. These must be active before you can load a recipe,
	// which is further down in the Initialization program.
	WHILE NOT(MpRecipeRegPar_PreviewPar.Active OR MpRecipeRegPar_PreviewPar.Error) DO
		MpRecipeRegPar_PreviewPar();
	END_WHILE
	WHILE NOT(MpRecipeRegPar_PreviewCfg.Active OR MpRecipeRegPar_PreviewCfg.Error) DO
		MpRecipeRegPar_PreviewCfg();
	END_WHILE

	// Load default Machine Settings recipe
	HmiRecipe.Parameters.Category := MACHINE_CONFIGURATION_CATEGORY;
	HmiRecipe.Parameters.FileName := DEFAULT_MACHINE_CONFIGURATION;
	MpRecipe_0.Load := TRUE;
	WHILE NOT(MpRecipe_0.CommandDone OR MpRecipe_0.Error) DO
		MpRecipe_0();
    END_WHILE
	MachineSettings := MachineSettingsPreview;

	MpRecipe_0.ErrorReset := MpRecipe_0.Error;
	MpRecipe_0.Load := FALSE;
	MpRecipe_0();

	// Load default Parameter recipe
	HmiRecipe.Parameters.Category := PARAMETERS_CATEGORY;
	HmiRecipe.Parameters.FileName := DEFAULT_PARAMETERS;
	HmiRecipe.Status.PreviousRecipe := DEFAULT_PARAMETERS;
	MpRecipe_0.Load := TRUE;
	WHILE NOT(MpRecipe_0.CommandDone OR MpRecipe_0.Error) DO
		MpRecipe_0();
	END_WHILE
	Parameters := ParametersPreview;

	HmiRecipe.Status.LastLoadedProductRecipe := DEFAULT_PARAMETERS;
	HmiRecipe.Status.LastLoadedConfigRecipe := DEFAULT_MACHINE_CONFIGURATION;
	MpRecipe_0.ErrorReset := MpRecipe_0.Error;
	MpRecipe_0.Load := FALSE;
	MpRecipe_0();

    // Trigger update notification so that the initial parameters are copied to the process
    // might not be necessary.*****
	MpRecipe_0.UpdateNotification := TRUE;

	// Init Filemanager for exporting/importing files
	MpFileManagerUI_0.Enable := TRUE;
	MpFileManagerUI_0.MpLink := ADR(gMpLinkFileManagerUIRecipe);
	MpFileManagerUI_0.UIConnect := ADR(MpFileManagerUIConnect);
	MpFileManagerUI_0.UISetup.FileListSize := SIZEOF(MpFileManagerUIConnect.File.List.Items) / SIZEOF(MpFileManagerUIConnect.File.List.Items[0]);
	MpFileManagerUIConnect.DeviceList.DeviceNames[0] := 'mappRecipeFiles';
	MpFileManagerUIConnect.DeviceList.DeviceNames[1] := '';
	MpFileManagerUI_0();

	HmiRecipe.Status.HMIcommand := REC_HMI_WAIT;

END_PROGRAM

PROGRAM _CYCLIC

	// Call actions
	FormatDeviceDataProvider;
	LoadPreview;
	RecipeHMIcommands;
	FileCopyOperation;

	// Reset commands on MpRecipe FUB
	IF MpRecipe_0.CommandDone THEN
		MpRecipe_0.Load := FALSE;
		MpRecipe_0.Save := FALSE;
		// Set update notification for machine category
	//	IF ((brsstrcmp(ADR(HmiRecipe.Parameters.Category), ADR(MACHINE_CONFIGURATION_CATEGORY)) = 0) AND (MpRecipe_0.Save = TRUE)) THEN
		IF ((brsstrcmp(ADR(HmiRecipe.Status.CategoryDropdown), ADR(MACHINE_CONFIGURATION_CATEGORY)) = 0) AND (MpRecipe_0.Save = TRUE)) THEN
			MpRecipe_0.UpdateNotification := TRUE;
		ELSE
			MpRecipe_0.UpdateNotification := FALSE;
			HmiRecipe.Parameters.Category := PARAMETERS_CATEGORY;
			HmiRecipe.Parameters.FileName := 'Default.par';
		END_IF
		END_IF

	// Error reset
	IF NOT MpRecipe_0.Error THEN
		MpRecipe_0.ErrorReset := FALSE;
	END_IF

	IF NOT MpRecipeUI_0.Error THEN
		MpRecipeUI_0.ErrorReset := FALSE;
	END_IF

	// Assign MpLinks
	MpRecipe_0.MpLink := ADR(gMpLinkRecipeXml);
	MpRecipeUI_0.MpLink := ADR(gMpLinkRecipeXml);
	MpFileManagerUI_0.MpLink := ADR(gMpLinkFileManagerUIRecipe);
	MpRecipeRegPar_PreviewPar.MpLink := ADR(gMpLinkRecipeXml);
	MpRecipeRegPar_PreviewCfg.MpLink := ADR(gMpLinkRecipeXml);

	// Call function blocks
	MpRecipe_0();
	MpRecipeUI_0();
	MpFileManagerUI_0();
	MpRecipeRegPar_PreviewPar();
	MpRecipeRegPar_PreviewCfg();

END_PROGRAM

PROGRAM _EXIT

	// Disable the function blocls to unlink the MpLinks
	MpRecipe_0.Enable := FALSE;
	MpRecipeUI_0.Enable := FALSE;
	MpRecipeRegPar_PreviewPar.Enable := FALSE;
	MpRecipeRegPar_PreviewCfg.Enable := FALSE;
	MpFileManagerUI_0.Enable := FALSE;

	// Call function blocks
	MpRecipe_0();
	MpRecipeUI_0();
	MpRecipeRegPar_PreviewPar();
	MpRecipeRegPar_PreviewCfg();
	MpFileManagerUI_0();

END_PROGRAM
```

#### RecipeMgr.typ - Local data types
```iecst
(*Structure types*)

TYPE
	RecipeHmiInterfaceType : 	STRUCT  (*Structure to hold commands, parameters and status from the HMI*)
		Commands : RecipeCommandsType; (*Structure to hold the commands from the HMI*)
		Parameters : RecipeParametersType; (*Structure to hold the parameters for the HMI*)
		Status : RecipeStatusType; (*Structure to hold status information from the mapp View HMI*)
	END_STRUCT;
	RecipeCommandsType : 	STRUCT  (*Structure to hold the commands from the HMI*)
		LoadRecipe : BOOL; (*Load recipe*)
		SaveSelectedRecipe : BOOL; (*Save the selected recipe (which is not necessarily the active recipe)*)
		CreateRecipe : BOOL; (*Create recipe*)
		ImportFromUSB : BOOL; (*Import from USB device*)
		ExportToUSB : BOOL; (*Export to USB device*)
	END_STRUCT;
	RecipeParametersType : 	STRUCT  (*Structure to hold the parameters for the HMI*)
		Category : STRING[30]; (*Current category*)
		DeviceDataProvider : ARRAY[0..MAX_IDX_FILE_DEV]OF STRING[100]; (*File device data provider*)
		DeviceName : STRING[50]; (*Selected file device name*)
		FileName : STRING[255]; (*Recipe file name*)
		TableConfig : STRING[120]; (*Table configuration *)
	END_STRUCT;
	RecipeStatusType : 	STRUCT  (*Structure to hold status information from the mapp View HMI*)
		HMIcommand : RecipeHmiStepEnum; (*State machine step for HMI commands*)
		LastLoadedConfigRecipe : STRING[255]; (*Last loaded configuration recipe*)
		LastLoadedProductRecipe : STRING[255]; (*Last loaded product recipe*)
		ActiveRecipe : STRING[255]; (*The name of the active recipe*)
		LastSelectedIndex : UINT; (*The previous selected index*)
		LastStatus : MpRecipeUIStatusEnum; (*The previous UI status*)
		CopyStep : RecipeCopyStepEnum; (*State machine step for copying a recipe to/from a USB drive*)
		CategoryDropdown : STRING[50]; (*Category dropdown value*)
		EditDialogOpened : BOOL; (*Flag that the edit dialog box was opened*)
		CreateDialogOpened : BOOL; (*Flag that the create dialog box was opened*)
		PreviousRecipe : STRING[80]; (*Name of the previous recipe*)
		FileDuplicate : BOOL; (*Recipe file already exists, warn the user.*)
		FilesAvailable : BOOL; (*Control access to widget when no files are available*)
	END_STRUCT;
	ParametersType : 	STRUCT  (*Demo / starter structure for machine parameters*)
		AddParametersHere1 : BOOL; (*Add your parameteres here *)
		AddParametersHere2 : STRING[80]; (*Add your parameteres here *)
		AddParametersHere3 : REAL; (*Add your parameteres here *)
		AddParametersHere4 : REAL; (*Add your parameteres here *)
		AddParametersHere5 : REAL; (*Add your parameteres here *)
	END_STRUCT;
	MachineSettingsType : 	STRUCT  (*Demo / starter structure for machine configuration settings*)
		AddMachineSettingsHere1 : USINT; (*Add your settings here*)
		AddMachineSettingsHere2 : DINT; (*Add your settings here*)
		AddMachineSettingsHere3 : BOOL; (*Add your settings here*)
		AddMachineSettingsHere4 : REAL; (*Add your settings here*)
		AddMachineSettingsHere5 : UINT; (*Add your settings here*)
	END_STRUCT;
END_TYPE

(*Enumerations*)

TYPE
	RecipeCopyStepEnum :
		( (*State machine step for copying a recipe to/from a USB drive*)
		REC_COPY_WAIT := 0, (*Wait state*)
		REC_COPY_TO_USB, (*Copy to USB*)
		REC_COPY_FROM_USB, (*Copy from USB*)
		REC_COPY_BUSY (*Busy*)
		);
	RecipeHmiStepEnum :
		( (*State machine step for HMI commands*)
		REC_HMI_WAIT, (*Wait*)
		REC_HMI_LOAD, (*Load recipe*)
		REC_HMI_SAVE, (*Save recipe*)
		REC_HMI_CREATE (*Create recipe*)
		);
END_TYPE
```

#### RecipeMgr.var - Local variables
```iecst
(*Function Blocks*)
VAR
	MpRecipe_0 : MpRecipeXml; (*MpRecipe instance*)
	MpRecipeRegPar_PreviewPar : MpRecipeRegPar; (*MpRecipeRegPar instance for ParametersPreview variable*)
	MpRecipeRegPar_PreviewCfg : MpRecipeRegPar; (*MpRecipeRegPar instance for MachineSettingsPreview*)
	MpRecipeUI_0 : MpRecipeUI; (*MpRecupeUI instance*)
	MpFileManagerUI_0 : MpFileManagerUI; (*MpFileManagerUI instance*)
	DTGetTime_0 : DTGetTime; (*DTGetTime instance*)
	DirCreate_0 : DirCreate; (*DirCreate instance*)
END_VAR
(*Constants*)
VAR CONSTANT
	MAX_IDX_FILE_DEV : USINT := MAX_IDX_USB_DEV_LIST + 1; (*Maximum number of  file devices *)
	DEFAULT_PARAMETERS : STRING[12] := 'Default.par'; (*Default parameters recipe file name*)
	DEFAULT_MACHINE_CONFIGURATION : STRING[12] := 'Machine.mcfg'; (*Default machine configuration recipe file name*)
END_VAR
VAR
	PARAMETERS_RECIPE : STRING[50] := 'Parameters'; (*Value of the DropDownBox selection for the Parameters category*)
	MACHINE_CONFIGURATION_RECIPE : STRING[50] := 'Machine Configuration'; (*Value of the DropDownBox selection for the Machine Configuration category*)
END_VAR
VAR CONSTANT
	LOCAL_FOLDER : STRING[10] := 'Recipe'; (*Folder name on the file device for Recipe files*)
END_VAR
(*Structure Types*)
VAR
	HmiRecipe : RecipeHmiInterfaceType; (*HMI interface structure*)
	Parameters : ParametersType; (*Machine parameters. Used by the machine at runtime*)
	ParametersEdit : {REDUND_UNREPLICABLE} ParametersType; (*Machine parameters edit structure. Enables you to edit a recipe that is not currently active*)
	ParametersPreview : ParametersType; (*Machine parameters preview structure. Registered to the recipe. Enables you to preview a recipe that is not currently active.*)
	MachineSettings : MachineSettingsType; (*Machine settings. Used by the machine at runtime.*)
	MachineSettingsEdit : MachineSettingsType; (*Machine settings edit structure. Enables you to edit a recipe that is not currently active*)
	MachineSettingsPreview : MachineSettingsType; (*Machine settings preview structure. Registered to the recipe. Enables you to preview a recipe that is not currently active. *)
	MpRecipeUIConnect : MpRecipeUIConnectType; (*MpRecipeUI connection to the HMI*) (*ParameterFileStep : INT;*)
	MpRecipeUISetup : MpRecipeUISetupType; (*MpRecipeUI setup connection to the HMI*) (*ParameterFileStep : INT;*)
	MpFileManagerUIConnect : MpFileManagerUIConnectType; (*File manager connection to the HMI*)
	Header : MpRecipeXmlHeaderType; (*Header information*)
END_VAR
(*Variables*)
VAR
	i : USINT; (*Index to loop through file devices*)
END_VAR
```

#### HMIActions.st - Supporting code for the HMI interface
```iecst
ACTION FormatDeviceDataProvider:

	// Select CF device if USB device is not available
	FOR i := 0 TO MAX_IDX_USB_DEV_LIST DO
		IF gUSBAvailable[i] THEN
			HmiRecipe.Parameters.DeviceDataProvider[i + 1] := '{"value":"USB';
			brsitoa(i + 1, ADR(HmiRecipe.Parameters.DeviceDataProvider[i + 1]) + brsstrlen(ADR(HmiRecipe.Parameters.DeviceDataProvider[i + 1])));
			brsstrcat(ADR(HmiRecipe.Parameters.DeviceDataProvider[i + 1]), ADR('","text":"USB'));
			brsitoa(i + 1, ADR(HmiRecipe.Parameters.DeviceDataProvider[i + 1]) + brsstrlen(ADR(HmiRecipe.Parameters.DeviceDataProvider[i + 1])));
			brsstrcat(ADR(HmiRecipe.Parameters.DeviceDataProvider[i + 1]), ADR('"}'));
			MpFileManagerUIConnect.DeviceList.DeviceNames[i + 1] := 'USB';
			brsitoa(i + 1, ADR(MpFileManagerUIConnect.DeviceList.DeviceNames[i + 1]) + brsstrlen(ADR(MpFileManagerUIConnect.DeviceList.DeviceNames[i + 1])));
		ELSE
			brsmemset(ADR(HmiRecipe.Parameters.DeviceDataProvider[i + 1]), 0, SIZEOF(HmiRecipe.Parameters.DeviceDataProvider[i + 1]));
			brsmemset(ADR(MpFileManagerUIConnect.DeviceList.DeviceNames[i + 1]), 0, SIZEOF(MpFileManagerUIConnect.DeviceList.DeviceNames[i + 1]));
		END_IF
	END_FOR

	// Configure visible recipe list
	IF MpRecipeUIConnect.Recipe.List.Names[0] = '' THEN
		HmiRecipe.Parameters.TableConfig := '{ "specRows": [{"from":0,"to":19, "visible":false}]}';
	ELSE
		HmiRecipe.Parameters.TableConfig := '{ "specRows": [{"from":';
		brsitoa(MpRecipeUIConnect.Recipe.List.MaxSelection + 1, ADR(HmiRecipe.Parameters.TableConfig) + brsstrlen(ADR(HmiRecipe.Parameters.TableConfig)));
		brsstrcat(ADR(HmiRecipe.Parameters.TableConfig),  ADR(',"to":19, "visible":false}]}'));
    END_IF

	HmiRecipe.Status.FilesAvailable := (MpRecipeUIConnect.Recipe.List.Names[0] <> '');

END_ACTION

ACTION LoadPreview:

	// Load preview when a recipe is selected
	IF (MpRecipeUIConnect.Recipe.List.SelectedIndex <> HmiRecipe.Status.LastSelectedIndex) OR (HmiRecipe.Status.LastMaxSelection <> MpRecipeUIConnect.Recipe.List.MaxSelection) THEN
		// Check selected recipe name is not empty
		IF (brsstrlen(ADR(MpRecipeUIConnect.Recipe.List.Names[MpRecipeUIConnect.Recipe.List.SelectedIndex])) > 0) THEN
			MpRecipe_0.FileName := ADR(MpRecipeUIConnect.Recipe.List.Names[MpRecipeUIConnect.Recipe.List.SelectedIndex]);
			MpRecipe_0.Category := ADR(HmiRecipe.Status.CategoryDropdown);
			MpRecipe_0.Load := TRUE;
			HmiRecipe.Status.LastSelectedIndex := MpRecipeUIConnect.Recipe.List.SelectedIndex;
			HmiRecipe.Status.LastMaxSelection := MpRecipeUIConnect.Recipe.List.MaxSelection;
		END_IF
	END_IF

	// Reset load command on MpRecipe_Pre FUB
	IF ((MpRecipe_0.CommandDone = TRUE) OR (MpRecipe_0.Error = TRUE)) THEN
		MpRecipe_0.Load := FALSE;
	END_IF

END_ACTION

ACTION RecipeHMIcommands:

	CASE HmiRecipe.Status.HMIcommand OF
		REC_HMI_WAIT:
			// The following commands are triggered directly from the HMI. If you imported the mapp View front end of
			// the Framework, then this is already taken care of. If you did not, then your visualization must
			// trigger each one of these command variables (CreateRecipe, SaveSelectedRecipe, LoadRecipe).
			IF HmiRecipe.Commands.CreateRecipe THEN
				HmiRecipe.Status.HMIcommand := REC_HMI_CREATE;
				HmiRecipe.Commands.CreateRecipe := FALSE;
			ELSIF HmiRecipe.Commands.SaveSelectedRecipe THEN
				HmiRecipe.Status.HMIcommand := REC_HMI_SAVE;
				HmiRecipe.Commands.SaveSelectedRecipe := FALSE;
			ELSIF HmiRecipe.Commands.LoadRecipe THEN
				HmiRecipe.Status.HMIcommand := REC_HMI_LOAD;
				HmiRecipe.Commands.LoadRecipe := FALSE;
			END_IF

		REC_HMI_CREATE:
			IF (brsstrcmp(ADR(HmiRecipe.Status.CategoryDropdown), ADR(PARAMETERS_RECIPE)) = 0) THEN
				ParametersPreview := ParametersEdit;
				brsstrcat(ADR(MpRecipeUIConnect.New.FileName),ADR('.par'));
			ELSIF (brsstrcmp(ADR(HmiRecipe.Status.CategoryDropdown), ADR(MACHINE_CONFIGURATION_RECIPE)) = 0) THEN
				MachineSettingsPreview := MachineSettingsEdit;
				brsstrcat(ADR(MpRecipeUIConnect.New.FileName),ADR('.mcfg'));
			END_IF

			Header.Name := MpRecipeUIConnect.New.FileName;
			DTGetTime_0.enable := TRUE;
			DTGetTime_0();
			WHILE DTGetTime_0.status <> 0 DO
				DTGetTime_0();
			END_WHILE;
			Header.DateTime := DTGetTime_0.DT1;
			DTGetTime_0.enable := FALSE;
			DTGetTime_0();
			MpRecipeUIConnect.New.Create := TRUE;
			HmiRecipe.Status.HMIcommand := REC_HMI_WAIT;

		REC_HMI_LOAD:
			IF (brsstrcmp(ADR(HmiRecipe.Status.CategoryDropdown), ADR(PARAMETERS_RECIPE)) = 0) THEN
				Parameters := ParametersPreview;
				HmiRecipe.Status.LastLoadedProductRecipe := HmiRecipe.Status.ActiveRecipe;
			ELSIF (brsstrcmp(ADR(HmiRecipe.Status.CategoryDropdown), ADR(MACHINE_CONFIGURATION_RECIPE)) = 0) THEN
				MachineSettings := MachineSettingsPreview;
				HmiRecipe.Status.LastLoadedConfigRecipe := HmiRecipe.Status.ActiveRecipe;
			END_IF
			HmiRecipe.Status.HMIcommand := REC_HMI_WAIT;

		REC_HMI_SAVE:
			IF (brsstrcmp(ADR(HmiRecipe.Status.CategoryDropdown), ADR(PARAMETERS_RECIPE)) = 0) THEN
				ParametersPreview := ParametersEdit;
	        ELSIF (brsstrcmp(ADR(HmiRecipe.Status.CategoryDropdown), ADR(MACHINE_CONFIGURATION_RECIPE)) = 0) THEN
                MachineSettingsPreview := MachineSettingsEdit;
            END_IF

			IF (brsstrlen(ADR(HmiRecipe.Status.ActiveRecipe)) > 0) THEN
				MpRecipe_0.FileName := ADR(HmiRecipe.Status.ActiveRecipe);
				MpRecipe_0.Save := TRUE;
			END_IF
			HmiRecipe.Status.HMIcommand := REC_HMI_WAIT;

	END_CASE

	IF NOT MpRecipe_0.CommandBusy AND brsstrcmp(ADR(HmiRecipe.Status.PreviousRecipe), ADR(HmiRecipe.Parameters.FileName)) <> 0 THEN
		HmiRecipe.Parameters.FileName := HmiRecipe.Status.PreviousRecipe;
	END_IF

	// If the Edit or Create dialog boxes open, copy the Preview structure into the Edit structure.
	IF HmiRecipe.Status.EditDialogOpened OR HmiRecipe.Status.CreateDialogOpened THEN
		IF (brsstrcmp(ADR(HmiRecipe.Status.CategoryDropdown), ADR(PARAMETERS_RECIPE)) = 0) THEN
			ParametersEdit := ParametersPreview;
			MpRecipeUIConnect.New.FileName := 'newParameters';
		ELSIF (brsstrcmp(ADR(HmiRecipe.Status.CategoryDropdown), ADR(MACHINE_CONFIGURATION_RECIPE)) = 0) THEN
			MachineSettingsEdit := MachineSettingsPreview;
			MpRecipeUIConnect.New.FileName := 'newMachConfig';
		END_IF

		HmiRecipe.Status.EditDialogOpened := FALSE;
		HmiRecipe.Status.CreateDialogOpened := FALSE;
	END_IF

	HmiRecipe.Status.FileDuplicate := FALSE;
	FOR i:= 0 TO 19 DO
		temp := MpRecipeUIConnect.New.FileName;
		IF (brsstrcmp(ADR(HmiRecipe.Status.CategoryDropdown), ADR(PARAMETERS_RECIPE)) = 0) THEN
			brsstrcat(ADR(temp),ADR('.par'));
		ELSIF (brsstrcmp(ADR(HmiRecipe.Status.CategoryDropdown), ADR(MACHINE_CONFIGURATION_RECIPE)) = 0) THEN
			brsstrcat(ADR(temp),ADR('.mcfg'));
		END_IF
		IF temp = MpRecipeUIConnect.Recipe.List.Names[i] THEN
			HmiRecipe.Status.FileDuplicate := TRUE;
		END_IF
	END_FOR

	HmiRecipe.Status.LastStatus := MpRecipeUIConnect.Status;
	HmiRecipe.Status.ActiveRecipe := MpRecipeUIConnect.Recipe.List.Names[MpRecipeUIConnect.Recipe.List.SelectedIndex];

END_ACTION
```

#### FileOperations.st - Handles copying recipes between User partition and USB stick
```iecst
ACTION FileCopyOperation:

	// Export/Import recipes to/from USB
    CASE HmiRecipe.Status.CopyStep OF
		REC_COPY_WAIT:
			// Wait for export/import command
            IF (HmiRecipe.Commands.ExportToUSB = TRUE) THEN
                // Check if USB device is available
                IF (brsstrlen(ADR(MpFileManagerUIConnect.DeviceList.DeviceNames[1])) > 0) THEN
					// USB is available proceed with export: select all files on the CF and trigger copy command
                    IF (MpFileManagerUIConnect.DeviceList.SelectedIndex <> 0) THEN
                        MpFileManagerUIConnect.DeviceList.SelectedIndex := 0;
                        MpFileManagerUIConnect.File.MultiSelect := FALSE;
                    ELSIF (MpFileManagerUIConnect.Status = mpFILE_UI_STATUS_IDLE) THEN

                        IF NOT MpFileManagerUIConnect.File.MultiSelect THEN
                            MpFileManagerUIConnect.File.MultiSelect := TRUE;
                            FOR i := 0 TO 49 DO
                                MpFileManagerUIConnect.File.List.Items[i].IsSelected := TRUE;
                            END_FOR
                        ELSIF (brsstrlen(ADR(MpFileManagerUIConnect.File.List.Items[i].Name)) = 0) THEN
                            // No files to copy, cancel operation
                            HmiRecipe.Commands.ExportToUSB := FALSE;
                        ELSE
                            MpFileManagerUIConnect.File.Copy := TRUE;
							HmiRecipe.Status.CopyStep := REC_COPY_TO_USB;
                            HmiRecipe.Commands.ExportToUSB := FALSE;
                        END_IF

                    END_IF

                ELSE
                    // No USB disk available, cancel operation
                    HmiRecipe.Commands.ExportToUSB := FALSE;
                END_IF

            ELSIF HmiRecipe.Commands.ImportFromUSB THEN
                // Check if USB device is available
                IF (brsstrlen(ADR(MpFileManagerUIConnect.DeviceList.DeviceNames[1])) > 0) THEN
                    // USB is available proceed with import: select all files on the USB and trigger copy command

                    IF (MpFileManagerUIConnect.DeviceList.SelectedIndex <> 1) THEN
                        MpFileManagerUIConnect.DeviceList.SelectedIndex := 1;
                        MpFileManagerUIConnect.File.MultiSelect := FALSE;
                    ELSIF MpFileManagerUIConnect.Status = mpFILE_UI_STATUS_IDLE THEN

                        IF NOT MpFileManagerUIConnect.File.MultiSelect THEN
                            MpFileManagerUIConnect.File.MultiSelect := TRUE;
                            FOR i := 0 TO ((SIZEOF(MpFileManagerUIConnect.File.List.Items)/SIZEOF(MpFileManagerUIConnect.File.List.Items[0])) - 1) DO
                                MpFileManagerUIConnect.File.List.Items[i].IsSelected := TRUE;
                            END_FOR
                        ELSIF (brsstrlen(ADR(MpFileManagerUIConnect.File.List.Items[i].Name)) = 0) THEN
                            // No files to copy, cancel operation
                            HmiRecipe.Commands.ImportFromUSB := FALSE;
                        ELSE
                            MpFileManagerUIConnect.File.Copy := TRUE;
                            HmiRecipe.Status.CopyStep := REC_COPY_FROM_USB;
                            HmiRecipe.Commands.ImportFromUSB := FALSE;
                        END_IF

                    END_IF
                ELSE
                    // No USB disk available, cancel operation
                    HmiRecipe.Commands.ImportFromUSB := FALSE;
                END_IF

            END_IF

		REC_COPY_TO_USB:
			// Navigate to USB device and paste files
            IF (MpFileManagerUIConnect.Status = mpFILE_UI_STATUS_IDLE) THEN

                IF (MpFileManagerUIConnect.DeviceList.SelectedIndex <> 1) THEN
                    MpFileManagerUIConnect.DeviceList.SelectedIndex := 1;
                    MpFileManagerUIConnect.File.MultiSelect := FALSE;
                ELSE
                    MpFileManagerUIConnect.File.Paste := TRUE;
                END_IF

            END_IF

            IF MpFileManagerUIConnect.Status = mpFILE_UI_STATUS_PASTE THEN
                HmiRecipe.Status.CopyStep := REC_COPY_BUSY;
            END_IF

		REC_COPY_FROM_USB:
			// Navigate to CF device and paste files
            IF (MpFileManagerUIConnect.DeviceList.SelectedIndex <> 0) THEN
                MpFileManagerUIConnect.DeviceList.SelectedIndex := 0;
                MpFileManagerUIConnect.File.MultiSelect := FALSE;
            ELSIF (MpFileManagerUIConnect.Status = mpFILE_UI_STATUS_IDLE) THEN
                MpFileManagerUIConnect.File.Paste := TRUE;
            END_IF

            IF (MpFileManagerUIConnect.Status = mpFILE_UI_STATUS_PASTE) THEN
                HmiRecipe.Status.CopyStep := REC_COPY_BUSY;
            END_IF

		REC_COPY_BUSY:
			// Wait for copying done
            IF (MpFileManagerUIConnect.MessageBox.Type = mpFILE_MSG_CONFIRM_OVERWRITE) OR (MpFileManagerUIConnect.MessageBox.Type = mpFILE_MSG_BUSY) THEN
                // TODO: Replace by confirm dialog
                MpFileManagerUIConnect.MessageBox.Confirm := TRUE;
            ELSIF MpFileManagerUIConnect.Status = mpFILE_UI_STATUS_IDLE THEN
                MpRecipeUIConnect.Recipe.Refresh := (MpRecipeUIConnect.Status = mpRECIPE_UI_STATUS_IDLE);
                HmiRecipe.Status.CopyStep := REC_COPY_WAIT;
            END_IF

    END_CASE

END_ACTION
```

#### RecipeMgt.st - not listed in the package file held
```iecst
//***********************************************************************
// Copyright: B&R Industrial Automation GmbH
// Author: B&R Industrial Automation GmbH
// Created: Jan 1, 2022
// Description: Tasks for recipe control.
//***********************************************************************

PROGRAM _INIT

	// Create folder for this component on the user file device
	DirCreate_New(enable := TRUE, pDevice := ADR('userPartition'), pName := ADR(LOCAL_FOLDER));

	// Check if folder already exist and if so disabled the function block call
	IF DirCreate_New.status = fiERR_DIR_ALREADY_EXIST THEN
		DirCreate_New(enable := FALSE);
	END_IF

	// Initialize mapp function blocks
	MpRecipeUISetup.Confirmation.RecipeDelete := TRUE;
	MpRecipeUISetup.RecipeListSize := 10;
	MpRecipeUISetup.RecipeListScrollWindow := 0;
	MpRecipeUISetup.AutoLoadHeader := TRUE;
	MpRecipeUIConnect.New.FileName := 'newRecipe.par';
	MpRecipeUIConnect.Recipe.Filter := '*par';
	MpRecipeUI_0.MpLink := ADR(gMpLinkRecipeXml);
	MpRecipeUI_0.Enable := TRUE;
	MpRecipeUI_0.UIConnect := ADR(MpRecipeUIConnect);
	MpRecipeUI_0.UISetup := MpRecipeUISetup;
	MpRecipeUI_0();

	HmiRecipe.Parameters.Category := PRODUCT_CATEGORY;
	HmiRecipe.Parameters.DeviceDataProvider[0] := '{"value":"mappRecipeFiles","text":"CF/PLC"}';
	HmiRecipe.Parameters.DeviceName := 'mappRecipeFiles';
	MpRecipe_0.MpLink := ADR(gMpLinkRecipeXml);
	MpRecipe_0.Enable := TRUE;
	MpRecipe_0.Category := ADR(HmiRecipe.Parameters.Category);
	MpRecipe_0.DeviceName := ADR(HmiRecipe.Parameters.DeviceName);
    MpRecipe_0.FileName := ADR(HmiRecipe.Parameters.FileName);
	MpRecipe_0.Header := ADR(Header);

	// Wait for MpRecipe_0 to activate. This must be active before you can call the RegPar function blocks,
	// which is further down in the Initialization program.
	WHILE NOT(MpRecipe_0.Active OR MpRecipe_0.Error) DO
		MpRecipe_0();
	END_WHILE

    MpRecipeRegPar_PreviewPar.MpLink := ADR(gMpLinkRecipeXml);
	MpRecipeRegPar_PreviewPar.Enable := TRUE;
	MpRecipeRegPar_PreviewPar.PVName := ADR('RecipeMgr:ParametersPreview');
	MpRecipeRegPar_PreviewPar.Category := ADR(PRODUCT_CATEGORY);
	MpRecipeRegPar_PreviewPar();

	MpRecipeRegPar_PreviewCfg.MpLink := ADR(gMpLinkRecipeXml);
	MpRecipeRegPar_PreviewCfg.Enable := TRUE;
	MpRecipeRegPar_PreviewCfg.PVName := ADR('RecipeMgr:MachineSettingsPreview');
	MpRecipeRegPar_PreviewCfg.Category := ADR(MACHINE_CATEGORY);
	MpRecipeRegPar_PreviewCfg();

	// Wait for RegPar function blocks to activate. These must be active before you can load a recipe,
	// which is further down in the Initialization program.
	WHILE NOT(MpRecipeRegPar_PreviewPar.Active OR MpRecipeRegPar_PreviewPar.Error) DO
		MpRecipeRegPar_PreviewPar();
	END_WHILE
	WHILE NOT(MpRecipeRegPar_PreviewCfg.Active OR MpRecipeRegPar_PreviewCfg.Error) DO
		MpRecipeRegPar_PreviewCfg();
	END_WHILE

	// Load default Machine Settings recipe
	HmiRecipe.Parameters.Category := MACHINE_CATEGORY;
	HmiRecipe.Parameters.FileName := MACHINE_FILENAME;
	MpRecipe_0.Load := TRUE;
	WHILE NOT(MpRecipe_0.CommandDone OR MpRecipe_0.Error) DO
		MpRecipe_0();
    END_WHILE
	MachineSettings := MachineSettingsPreview;

	MpRecipe_0.ErrorReset := MpRecipe_0.Error;
	MpRecipe_0.Load := FALSE;
	MpRecipe_0();

	// Load default Parameter recipe
	HmiRecipe.Parameters.Category := PRODUCT_CATEGORY;
	HmiRecipe.Parameters.FileName := 'Default.par';
	PreviousRecipe := 'Default.par';
	MpRecipe_0.Load := TRUE;
	WHILE NOT(MpRecipe_0.CommandDone OR MpRecipe_0.Error) DO
		MpRecipe_0();
	END_WHILE
	Parameters := ParametersPreview;

	HmiRecipe.Parameters.LastLoadedProductRecipe := MpRecipe_0.Info.LastLoadedRecipe;
	HmiRecipe.Parameters.LastLoadedConfigRecipe := MACHINE_FILENAME;
	MpRecipe_0.ErrorReset := MpRecipe_0.Error;
	MpRecipe_0.Load := FALSE;
	MpRecipe_0();

    // Trigger update notification so that the initial parameters are copied to the process
    // might not be necessary.*****
	MpRecipe_0.UpdateNotification := TRUE;

	// Init Filemanager for exporting/importing files
	MpFileManagerUI_0.Enable := TRUE;
	MpFileManagerUI_0.MpLink := ADR(gMpLinkFileManagerUIRecipe);
	MpFileManagerUI_0.UIConnect := ADR(MpFileManagerUIConnect);
	MpFileManagerUI_0.UISetup.FileListSize := SIZEOF(MpFileManagerUIConnect.File.List.Items) / SIZEOF(MpFileManagerUIConnect.File.List.Items[0]);
	MpFileManagerUIConnect.DeviceList.DeviceNames[0] := 'mappRecipeFiles';
	MpFileManagerUIConnect.DeviceList.DeviceNames[1] := '';
	MpFileManagerUI_0();

	HmiRecipe.Status.HMIcommand := REC_HMI_WAIT;

END_PROGRAM

PROGRAM _CYCLIC

	// Call actions
	FormatDeviceDataProvider;
	LoadPreview;
	RecipeHMIcommands;
	FileCopyOperation;

    // Reset category after saving is done, category should be reset so that autosave files contain ALL the parameters
    IF EDGEPOS(MpRecipeUIConnect.Status = mpRECIPE_UI_STATUS_IDLE) AND ((NOT MpRecipeUIConnect.Recipe.Load) AND (NOT MpRecipeUIConnect.Recipe.Save)) THEN
        // Check if 'Product' category has been loaded
        IF ((brsstrcmp(ADR(HmiRecipe.Parameters.Category), ADR(PRODUCT_CATEGORY)) = 0) AND (HmiRecipe.Parameters.LastStatus = mpRECIPE_UI_STATUS_LOAD)) THEN
			HmiRecipe.Parameters.LastLoadedProductRecipe := MpRecipe_0.Info.LastLoadedRecipe;
			MpRecipe_0.UpdateNotification := TRUE;
		ELSIF ((brsstrcmp(ADR(HmiRecipe.Parameters.Category), ADR(MACHINE_CATEGORY)) = 0) AND (HmiRecipe.Parameters.LastStatus = mpRECIPE_UI_STATUS_LOAD)) THEN
			HmiRecipe.Parameters.LastLoadedConfigRecipe := MpRecipe_0.Info.LastLoadedRecipe;
			MpRecipe_0.UpdateNotification := TRUE;
        END_IF
		// Trigger a reload of the preview parameters
        HmiRecipe.Parameters.LastSelectedIndex := HmiRecipe.Parameters.LastSelectedIndex + 1;
        brsstrcpy(ADR(HmiRecipe.Parameters.Category), ADR(PRODUCT_CATEGORY));
    END_IF
    HmiRecipe.Parameters.LastStatus := MpRecipeUIConnect.Status;
	HmiRecipe.Parameters.ActiveRecipe := MpRecipeUIConnect.Recipe.List.Names[MpRecipeUIConnect.Recipe.List.SelectedIndex];

    // Save current recipe
    IF (HmiRecipe.Commands.SaveCurrentRecipe = TRUE) AND NOT (MpRecipe_0.Load OR MpRecipe_0.Save OR MpRecipe_0.UpdateNotification) THEN
		HmiRecipe.Parameters.FileName := HmiRecipe.Parameters.LastLoadedProductRecipe;
        DTGetTime_0(enable := TRUE);
        Header.DateTime := DTGetTime_0.DT1;
        Header.Name := HmiRecipe.Parameters.FileName;
        Header.Description := '';
        MpRecipe_0.Save := TRUE;
        HmiRecipe.Commands.SaveCurrentRecipe := FALSE;
    END_IF

	// Reset commands on MpRecipe FUB
	IF MpRecipe_0.CommandDone THEN
		// Set update notification for machine category
		IF ((brsstrcmp(ADR(HmiRecipe.Parameters.Category), ADR(MACHINE_CATEGORY)) = 0) AND (MpRecipe_0.Save = TRUE)) THEN
			MpRecipe_0.UpdateNotification := TRUE;
			MpRecipe_0.Load := FALSE;
			MpRecipe_0.Save := FALSE;
		ELSE
			MpRecipe_0.UpdateNotification := FALSE;
			MpRecipe_0.Load := FALSE;
			MpRecipe_0.Save := FALSE;
			HmiRecipe.Parameters.Category := PRODUCT_CATEGORY;
			HmiRecipe.Parameters.FileName := 'Default.par';
        END_IF
    END_IF

	// Error reset
	IF NOT MpRecipe_0.Error THEN
		MpRecipe_0.ErrorReset := FALSE;
	END_IF

	IF NOT MpRecipeUI_0.Error THEN
		MpRecipeUI_0.ErrorReset := FALSE;
	END_IF

	// Assign MpLinks
	MpRecipe_0.MpLink := ADR(gMpLinkRecipeXml);
	MpRecipeUI_0.MpLink := ADR(gMpLinkRecipeXml);
	MpFileManagerUI_0.MpLink := ADR(gMpLinkFileManagerUIRecipe);
	MpRecipeRegPar_PreviewPar.MpLink := ADR(gMpLinkRecipeXml);
	MpRecipeRegPar_PreviewCfg.MpLink := ADR(gMpLinkRecipeXml);

	// Call function blocks
	MpRecipe_0();
	MpRecipeUI_0();
	MpFileManagerUI_0();
	MpRecipeRegPar_PreviewPar();
	MpRecipeRegPar_PreviewCfg();

END_PROGRAM

PROGRAM _EXIT

	// Disable the function blocls to unlink the MpLinks
	MpRecipe_0.Enable := FALSE;
	MpRecipeUI_0.Enable := FALSE;
	MpRecipeRegPar_PreviewPar.Enable := FALSE;
	MpRecipeRegPar_PreviewCfg.Enable := FALSE;
	MpFileManagerUI_0.Enable := FALSE;

	// Call function blocks
	MpRecipe_0();
	MpRecipeUI_0();
	MpRecipeRegPar_PreviewPar();
	MpRecipeRegPar_PreviewCfg();
	MpFileManagerUI_0();

END_PROGRAM
```

### Program Logical/Infrastructure/Recipe/Recipe (IEC)

#### Recipe.st - Init, cyclic, exit code
```iecst
//***********************************************************************
// Copyright: B&R Industrial Automation GmbH
// Author: B&R Industrial Automation GmbH
// Created: Jan 1, 2022
// Description: Tasks for recipe control.
//***********************************************************************

PROGRAM _INIT

	// Create folder for this component on the user file device
	DirCreate_New(enable := TRUE, pDevice := ADR('userPartition'), pName := ADR(LOCAL_FOLDER));

	// Check if folder already exist and if so disabled the function block call
	IF DirCreate_New.status = fiERR_DIR_ALREADY_EXIST THEN
		DirCreate_New(enable := FALSE);
	END_IF

	// Initialize mapp function blocks
	MpRecipeUISetup.Confirmation.RecipeDelete := TRUE;
	MpRecipeUISetup.RecipeListSize := 10;
	MpRecipeUISetup.RecipeListScrollWindow := 0;
	MpRecipeUISetup.AutoLoadHeader := TRUE;
	MpRecipeUIConnect.New.FileName := 'newRecipe.par';
	MpRecipeUIConnect.Recipe.Filter := '*par';
	MpRecipeUI_0.MpLink := ADR(gMpLinkRecipeXml);
	MpRecipeUI_0.Enable := TRUE;
	MpRecipeUI_0.UIConnect := ADR(MpRecipeUIConnect);
	MpRecipeUI_0.UISetup := MpRecipeUISetup;
	MpRecipeUI_0();

	HmiRecipe.Parameters.Category := PRODUCT_CATEGORY;
	HmiRecipe.Parameters.DeviceDataProvider[0] := '{"value":"mappRecipeFiles","text":"CF/PLC"}';
	HmiRecipe.Parameters.DeviceName := 'mappRecipeFiles';
	MpRecipe_0.MpLink := ADR(gMpLinkRecipeXml);
	MpRecipe_0.Enable := TRUE;
	MpRecipe_0.Category := ADR(HmiRecipe.Parameters.Category);
	MpRecipe_0.DeviceName := ADR(HmiRecipe.Parameters.DeviceName);
    MpRecipe_0.FileName := ADR(HmiRecipe.Parameters.FileName);
	MpRecipe_0.Header := ADR(Header);

	// Wait for MpRecipe_0 to activate. This must be active before you can call the RegPar function blocks,
	// which is further down in the Initialization program.
	WHILE NOT(MpRecipe_0.Active OR MpRecipe_0.Error) DO
		MpRecipe_0();
	END_WHILE

    MpRecipeRegPar_PreviewPar.MpLink := ADR(gMpLinkRecipeXml);
	MpRecipeRegPar_PreviewPar.Enable := TRUE;
	MpRecipeRegPar_PreviewPar.PVName := ADR('Recipe:ParametersPreview');
	MpRecipeRegPar_PreviewPar.Category := ADR(PRODUCT_CATEGORY);
	MpRecipeRegPar_PreviewPar();

	MpRecipeRegPar_PreviewCfg.MpLink := ADR(gMpLinkRecipeXml);
	MpRecipeRegPar_PreviewCfg.Enable := TRUE;
	MpRecipeRegPar_PreviewCfg.PVName := ADR('Recipe:MachineSettingsPreview');
	MpRecipeRegPar_PreviewCfg.Category := ADR(MACHINE_CATEGORY);
	MpRecipeRegPar_PreviewCfg();

	// Wait for RegPar function blocks to activate. These must be active before you can load a recipe,
	// which is further down in the Initialization program.
	WHILE NOT(MpRecipeRegPar_PreviewPar.Active OR MpRecipeRegPar_PreviewPar.Error) DO
		MpRecipeRegPar_PreviewPar();
	END_WHILE
	WHILE NOT(MpRecipeRegPar_PreviewCfg.Active OR MpRecipeRegPar_PreviewCfg.Error) DO
		MpRecipeRegPar_PreviewCfg();
	END_WHILE

	// Load default Machine Settings recipe
	HmiRecipe.Parameters.Category := MACHINE_CATEGORY;
	HmiRecipe.Parameters.FileName := MACHINE_FILENAME;
	MpRecipe_0.Load := TRUE;
	WHILE NOT(MpRecipe_0.CommandDone OR MpRecipe_0.Error) DO
		MpRecipe_0();
    END_WHILE
	MachineSettings := MachineSettingsPreview;

	MpRecipe_0.ErrorReset := MpRecipe_0.Error;
	MpRecipe_0.Load := FALSE;
	MpRecipe_0();

	// Load default Parameter recipe
	HmiRecipe.Parameters.Category := PRODUCT_CATEGORY;
	HmiRecipe.Parameters.FileName := 'Default.par';
	PreviousRecipe := 'Default.par';
	MpRecipe_0.Load := TRUE;
	WHILE NOT(MpRecipe_0.CommandDone OR MpRecipe_0.Error) DO
		MpRecipe_0();
	END_WHILE
	Parameters := ParametersPreview;

	HmiRecipe.Parameters.LastLoadedProductRecipe := MpRecipe_0.Info.LastLoadedRecipe;
	HmiRecipe.Parameters.LastLoadedConfigRecipe := MACHINE_FILENAME;
	MpRecipe_0.ErrorReset := MpRecipe_0.Error;
	MpRecipe_0.Load := FALSE;
	MpRecipe_0();

    // Trigger update notification so that the initial parameters are copied to the process
    // might not be necessary.*****
	MpRecipe_0.UpdateNotification := TRUE;

	// Init Filemanager for exporting/importing files
	MpFileManagerUI_0.Enable := TRUE;
	MpFileManagerUI_0.MpLink := ADR(gMpLinkFileManagerUIRecipe);
	MpFileManagerUI_0.UIConnect := ADR(MpFileManagerUIConnect);
	MpFileManagerUI_0.UISetup.FileListSize := SIZEOF(MpFileManagerUIConnect.File.List.Items) / SIZEOF(MpFileManagerUIConnect.File.List.Items[0]);
	MpFileManagerUIConnect.DeviceList.DeviceNames[0] := 'mappRecipeFiles';
	MpFileManagerUIConnect.DeviceList.DeviceNames[1] := '';
	MpFileManagerUI_0();

	HmiRecipe.Status.HMIcommand := REC_HMI_WAIT;

END_PROGRAM

PROGRAM _CYCLIC

	// Call actions
	FormatDeviceDataProvider;
	LoadPreview;
	RecipeHMIcommands;
	FileCopyOperation;

    // Reset category after saving is done, category should be reset so that autosave files contain ALL the parameters
    IF EDGEPOS(MpRecipeUIConnect.Status = mpRECIPE_UI_STATUS_IDLE) AND ((NOT MpRecipeUIConnect.Recipe.Load) AND (NOT MpRecipeUIConnect.Recipe.Save)) THEN
        // Check if 'Product' category has been loaded
        IF ((brsstrcmp(ADR(HmiRecipe.Parameters.Category), ADR(PRODUCT_CATEGORY)) = 0) AND (HmiRecipe.Parameters.LastStatus = mpRECIPE_UI_STATUS_LOAD)) THEN
			HmiRecipe.Parameters.LastLoadedProductRecipe := MpRecipe_0.Info.LastLoadedRecipe;
			MpRecipe_0.UpdateNotification := TRUE;
		ELSIF ((brsstrcmp(ADR(HmiRecipe.Parameters.Category), ADR(MACHINE_CATEGORY)) = 0) AND (HmiRecipe.Parameters.LastStatus = mpRECIPE_UI_STATUS_LOAD)) THEN
			HmiRecipe.Parameters.LastLoadedConfigRecipe := MpRecipe_0.Info.LastLoadedRecipe;
			MpRecipe_0.UpdateNotification := TRUE;
        END_IF
		// Trigger a reload of the preview parameters
        HmiRecipe.Parameters.LastSelectedIndex := HmiRecipe.Parameters.LastSelectedIndex + 1;
        brsstrcpy(ADR(HmiRecipe.Parameters.Category), ADR(PRODUCT_CATEGORY));
    END_IF
    HmiRecipe.Parameters.LastStatus := MpRecipeUIConnect.Status;
	HmiRecipe.Parameters.ActiveRecipe := MpRecipeUIConnect.Recipe.List.Names[MpRecipeUIConnect.Recipe.List.SelectedIndex];

    // Save current recipe
    IF (HmiRecipe.Commands.SaveCurrentRecipe = TRUE) AND NOT (MpRecipe_0.Load OR MpRecipe_0.Save OR MpRecipe_0.UpdateNotification) THEN
		HmiRecipe.Parameters.FileName := HmiRecipe.Parameters.LastLoadedProductRecipe;
        DTGetTime_0(enable := TRUE);
        Header.DateTime := DTGetTime_0.DT1;
        Header.Name := HmiRecipe.Parameters.FileName;
        Header.Description := '';
        MpRecipe_0.Save := TRUE;
        HmiRecipe.Commands.SaveCurrentRecipe := FALSE;
    END_IF

	// Reset commands on MpRecipe FUB
	IF MpRecipe_0.CommandDone THEN
		// Set update notification for machine category
		IF ((brsstrcmp(ADR(HmiRecipe.Parameters.Category), ADR(MACHINE_CATEGORY)) = 0) AND (MpRecipe_0.Save = TRUE)) THEN
			MpRecipe_0.UpdateNotification := TRUE;
			MpRecipe_0.Load := FALSE;
			MpRecipe_0.Save := FALSE;
		ELSE
			MpRecipe_0.UpdateNotification := FALSE;
			MpRecipe_0.Load := FALSE;
			MpRecipe_0.Save := FALSE;
			HmiRecipe.Parameters.Category := PRODUCT_CATEGORY;
			HmiRecipe.Parameters.FileName := 'Default.par';
        END_IF
    END_IF

	// Error reset
	IF NOT MpRecipe_0.Error THEN
		MpRecipe_0.ErrorReset := FALSE;
	END_IF

	IF NOT MpRecipeUI_0.Error THEN
		MpRecipeUI_0.ErrorReset := FALSE;
	END_IF

	// Assign MpLinks
	MpRecipe_0.MpLink := ADR(gMpLinkRecipeXml);
	MpRecipeUI_0.MpLink := ADR(gMpLinkRecipeXml);
	MpFileManagerUI_0.MpLink := ADR(gMpLinkFileManagerUIRecipe);
	MpRecipeRegPar_PreviewPar.MpLink := ADR(gMpLinkRecipeXml);
	MpRecipeRegPar_PreviewCfg.MpLink := ADR(gMpLinkRecipeXml);

	// Call function blocks
	MpRecipe_0();
	MpRecipeUI_0();
	MpFileManagerUI_0();
	MpRecipeRegPar_PreviewPar();
	MpRecipeRegPar_PreviewCfg();

END_PROGRAM

PROGRAM _EXIT

	// Disable the function blocls to unlink the MpLinks
	MpRecipe_0.Enable := FALSE;
	MpRecipeUI_0.Enable := FALSE;
	MpRecipeRegPar_PreviewPar.Enable := FALSE;
	MpRecipeRegPar_PreviewCfg.Enable := FALSE;
	MpFileManagerUI_0.Enable := FALSE;

	// Call function blocks
	MpRecipe_0();
	MpRecipeUI_0();
	MpRecipeRegPar_PreviewPar();
	MpRecipeRegPar_PreviewCfg();
	MpFileManagerUI_0();

END_PROGRAM
```

#### Recipe.typ - Local data types
```iecst
TYPE
	RecipeCommandsType : 	STRUCT
		StoreMachineSettings : BOOL;
		FactoryResetMachineSettings : BOOL;
		SaveCurrentRecipe : BOOL;
		ImportFromUSB : BOOL;
		ExportToUSB : BOOL;
		SaveSelectedRecipe : BOOL;
		LoadRecipe : BOOL;
		CreateRecipe : BOOL;
	END_STRUCT;
	RecipeParametersType : 	STRUCT
		Category : STRING[30];
		LastLoadedConfigRecipe : STRING[255];
		LastLoadedProductRecipe : STRING[255];
		ActiveRecipe : STRING[255];
		DeviceDataProvider : ARRAY[0..MAX_IDX_FILE_DEV]OF STRING[100];
		DeviceName : STRING[50];
		FileName : STRING[255];
		LastSelectedIndex : UINT;
		LastStatus : MpRecipeUIStatusEnum;
		TableConfig : STRING[120];
		CopyStep : RecipeCopyStepEnum;
		CategoryDropdown : STRING[50];
		EditDialogOpened : BOOL;
		CreateDialogOpened : BOOL;
	END_STRUCT;
	RecipeStatusType : 	STRUCT
		HMIcommand : RecipeHmiStepEnum;
	END_STRUCT;
	RecipeHmiInterfaceType : 	STRUCT
		Commands : RecipeCommandsType;
		Parameters : RecipeParametersType;
		Status : RecipeStatusType;
	END_STRUCT;
	RecipeCopyStepEnum :
		(
		REC_COPY_WAIT := 0,
		REC_COPY_TO_USB,
		REC_COPY_FROM_USB,
		REC_COPY_BUSY
		);
	MachineSettingsType : 	STRUCT
		AddMachineSettingsHere1 : USINT;
		AddMachineSettingsHere2 : DINT;
		AddMachineSettingsHere3 : BOOL;
		AddMachineSettingsHere4 : REAL;
		AddMachineSettingsHere5 : UINT;
	END_STRUCT;
	ParametersType : 	STRUCT
		AddParametersHere1 : BOOL;
		AddParametersHere2 : STRING[80];
		AddParametersHere3 : REAL;
		AddParametersHere4 : REAL;
		AddParametersHere5 : REAL;
	END_STRUCT;
	RecipeHmiStepEnum :
		(
		REC_HMI_WAIT,
		REC_HMI_LOAD,
		REC_HMI_SAVE,
		REC_HMI_CREATE
		);
END_TYPE
```

#### FileOperations.st
```iecst
ACTION FileCopyOperation:

	// Export/Import recipes to/from USB
    CASE HmiRecipe.Parameters.CopyStep OF
		REC_COPY_WAIT:
			// Wait for export/import command
            IF (HmiRecipe.Commands.ExportToUSB = TRUE) THEN
                // Check if USB device is available
                IF (brsstrlen(ADR(MpFileManagerUIConnect.DeviceList.DeviceNames[1])) > 0) THEN
					// USB is available proceed with export: select all files on the CF and trigger copy command
                    IF (MpFileManagerUIConnect.DeviceList.SelectedIndex <> 0) THEN
                        MpFileManagerUIConnect.DeviceList.SelectedIndex := 0;
                        MpFileManagerUIConnect.File.MultiSelect := FALSE;
                    ELSIF (MpFileManagerUIConnect.Status = mpFILE_UI_STATUS_IDLE) THEN

                        IF NOT MpFileManagerUIConnect.File.MultiSelect THEN
                            MpFileManagerUIConnect.File.MultiSelect := TRUE;
                            FOR Index := 0 TO 49 DO
                                MpFileManagerUIConnect.File.List.Items[Index].IsSelected := TRUE;
                            END_FOR
                        ELSIF (brsstrlen(ADR(MpFileManagerUIConnect.File.List.Items[Index].Name)) = 0) THEN
                            // No files to copy, cancel operation
                            HmiRecipe.Commands.ExportToUSB := FALSE;
                        ELSE
                            MpFileManagerUIConnect.File.Copy := TRUE;
							HmiRecipe.Parameters.CopyStep := REC_COPY_TO_USB;
                            HmiRecipe.Commands.ExportToUSB := FALSE;
                        END_IF

                    END_IF

                ELSE
                    // No USB disk available, cancel operation
                    HmiRecipe.Commands.ExportToUSB := FALSE;
                END_IF

            ELSIF HmiRecipe.Commands.ImportFromUSB THEN
                // Check if USB device is available
                IF (brsstrlen(ADR(MpFileManagerUIConnect.DeviceList.DeviceNames[1])) > 0) THEN
                    // USB is available proceed with import: select all files on the USB and trigger copy command

                    IF (MpFileManagerUIConnect.DeviceList.SelectedIndex <> 1) THEN
                        MpFileManagerUIConnect.DeviceList.SelectedIndex := 1;
                        MpFileManagerUIConnect.File.MultiSelect := FALSE;
                    ELSIF MpFileManagerUIConnect.Status = mpFILE_UI_STATUS_IDLE THEN

                        IF NOT MpFileManagerUIConnect.File.MultiSelect THEN
                            MpFileManagerUIConnect.File.MultiSelect := TRUE;
                            FOR Index := 0 TO ((SIZEOF(MpFileManagerUIConnect.File.List.Items)/SIZEOF(MpFileManagerUIConnect.File.List.Items[0])) - 1) DO
                                MpFileManagerUIConnect.File.List.Items[Index].IsSelected := TRUE;
                            END_FOR
                        ELSIF (brsstrlen(ADR(MpFileManagerUIConnect.File.List.Items[Index].Name)) = 0) THEN
                            // No files to copy, cancel operation
                            HmiRecipe.Commands.ImportFromUSB := FALSE;
                        ELSE
                            MpFileManagerUIConnect.File.Copy := TRUE;
                            HmiRecipe.Parameters.CopyStep := REC_COPY_FROM_USB;
                            HmiRecipe.Commands.ImportFromUSB := FALSE;
                        END_IF

                    END_IF
                ELSE
                    // No USB disk available, cancel operation
                    HmiRecipe.Commands.ImportFromUSB := FALSE;
                END_IF

            END_IF

		REC_COPY_TO_USB:
			// Navigate to USB device and paste files
            IF (MpFileManagerUIConnect.Status = mpFILE_UI_STATUS_IDLE) THEN

                IF (MpFileManagerUIConnect.DeviceList.SelectedIndex <> 1) THEN
                    MpFileManagerUIConnect.DeviceList.SelectedIndex := 1;
                    MpFileManagerUIConnect.File.MultiSelect := FALSE;
                ELSE
                    MpFileManagerUIConnect.File.Paste := TRUE;
                END_IF

            END_IF

            IF MpFileManagerUIConnect.Status = mpFILE_UI_STATUS_PASTE THEN
                HmiRecipe.Parameters.CopyStep := REC_COPY_BUSY;
            END_IF

		REC_COPY_FROM_USB:
			// Navigate to CF device and paste files
            IF (MpFileManagerUIConnect.DeviceList.SelectedIndex <> 0) THEN
                MpFileManagerUIConnect.DeviceList.SelectedIndex := 0;
                MpFileManagerUIConnect.File.MultiSelect := FALSE;
            ELSIF (MpFileManagerUIConnect.Status = mpFILE_UI_STATUS_IDLE) THEN
                MpFileManagerUIConnect.File.Paste := TRUE;
            END_IF

            IF (MpFileManagerUIConnect.Status = mpFILE_UI_STATUS_PASTE) THEN
                HmiRecipe.Parameters.CopyStep := REC_COPY_BUSY;
            END_IF

		REC_COPY_BUSY:
			// Wait for copying done
            IF (MpFileManagerUIConnect.MessageBox.Type = mpFILE_MSG_CONFIRM_OVERWRITE) OR (MpFileManagerUIConnect.MessageBox.Type = mpFILE_MSG_BUSY) THEN
                // TODO: Replace by confirm dialog
                MpFileManagerUIConnect.MessageBox.Confirm := TRUE;
            ELSIF MpFileManagerUIConnect.Status = mpFILE_UI_STATUS_IDLE THEN
                MpRecipeUIConnect.Recipe.Refresh := (MpRecipeUIConnect.Status = mpRECIPE_UI_STATUS_IDLE);
                HmiRecipe.Parameters.CopyStep := REC_COPY_WAIT;
            END_IF

    END_CASE

END_ACTION
```

### Program Logical/Infrastructure/Recipe/RecipeMgt (IEC)

#### RecipeMgt.st - Init, cyclic, exit code
```iecst
//***********************************************************************
// Copyright: B&R Industrial Automation GmbH
// Author: B&R Industrial Automation GmbH
// Created: Jan 1, 2022
// Description: Tasks for recipe control.
//***********************************************************************

PROGRAM _INIT

	// Create folder for this component on the user file device
	DirCreate_New(enable := TRUE, pDevice := ADR('userPartition'), pName := ADR(LOCAL_FOLDER));

	// Check if folder already exist and if so disabled the function block call
	IF DirCreate_New.status = fiERR_DIR_ALREADY_EXIST THEN
		DirCreate_New(enable := FALSE);
	END_IF

	// Initialize mapp function blocks
	MpRecipeUISetup.Confirmation.RecipeDelete := TRUE;
	MpRecipeUISetup.RecipeListSize := 10;
	MpRecipeUISetup.RecipeListScrollWindow := 0;
	MpRecipeUISetup.AutoLoadHeader := TRUE;
	MpRecipeUIConnect.New.FileName := 'newRecipe.par';
	MpRecipeUIConnect.Recipe.Filter := '*par';
	MpRecipeUI_0.MpLink := ADR(gMpLinkRecipeXml);
	MpRecipeUI_0.Enable := TRUE;
	MpRecipeUI_0.UIConnect := ADR(MpRecipeUIConnect);
	MpRecipeUI_0.UISetup := MpRecipeUISetup;
	MpRecipeUI_0();

	HmiRecipe.Parameters.Category := PRODUCT_CATEGORY;
	HmiRecipe.Parameters.DeviceDataProvider[0] := '{"value":"mappRecipeFiles","text":"CF/PLC"}';
	HmiRecipe.Parameters.DeviceName := 'mappRecipeFiles';
	MpRecipe_0.MpLink := ADR(gMpLinkRecipeXml);
	MpRecipe_0.Enable := TRUE;
	MpRecipe_0.Category := ADR(HmiRecipe.Parameters.Category);
	MpRecipe_0.DeviceName := ADR(HmiRecipe.Parameters.DeviceName);
    MpRecipe_0.FileName := ADR(HmiRecipe.Parameters.FileName);
	MpRecipe_0.Header := ADR(Header);

	// Wait for MpRecipe_0 to activate. This must be active before you can call the RegPar function blocks,
	// which is further down in the Initialization program.
	WHILE NOT(MpRecipe_0.Active OR MpRecipe_0.Error) DO
		MpRecipe_0();
	END_WHILE

    MpRecipeRegPar_PreviewPar.MpLink := ADR(gMpLinkRecipeXml);
	MpRecipeRegPar_PreviewPar.Enable := TRUE;
	MpRecipeRegPar_PreviewPar.PVName := ADR('RecipeMgt:ParametersPreview');
	MpRecipeRegPar_PreviewPar.Category := ADR(PRODUCT_CATEGORY);
	MpRecipeRegPar_PreviewPar();

	MpRecipeRegPar_PreviewCfg.MpLink := ADR(gMpLinkRecipeXml);
	MpRecipeRegPar_PreviewCfg.Enable := TRUE;
	MpRecipeRegPar_PreviewCfg.PVName := ADR('RecipeMgt:MachineSettingsPreview');
	MpRecipeRegPar_PreviewCfg.Category := ADR(MACHINE_CATEGORY);
	MpRecipeRegPar_PreviewCfg();

	// Wait for RegPar function blocks to activate. These must be active before you can load a recipe,
	// which is further down in the Initialization program.
	WHILE NOT(MpRecipeRegPar_PreviewPar.Active OR MpRecipeRegPar_PreviewPar.Error) DO
		MpRecipeRegPar_PreviewPar();
	END_WHILE
	WHILE NOT(MpRecipeRegPar_PreviewCfg.Active OR MpRecipeRegPar_PreviewCfg.Error) DO
		MpRecipeRegPar_PreviewCfg();
	END_WHILE

	// Load default Machine Settings recipe
	HmiRecipe.Parameters.Category := MACHINE_CATEGORY;
	HmiRecipe.Parameters.FileName := MACHINE_FILENAME;
	MpRecipe_0.Load := TRUE;
	WHILE NOT(MpRecipe_0.CommandDone OR MpRecipe_0.Error) DO
		MpRecipe_0();
    END_WHILE
	MachineSettings := MachineSettingsPreview;

	MpRecipe_0.ErrorReset := MpRecipe_0.Error;
	MpRecipe_0.Load := FALSE;
	MpRecipe_0();

	// Load default Parameter recipe
	HmiRecipe.Parameters.Category := PRODUCT_CATEGORY;
	HmiRecipe.Parameters.FileName := 'Default.par';
	PreviousRecipe := 'Default.par';
	MpRecipe_0.Load := TRUE;
	WHILE NOT(MpRecipe_0.CommandDone OR MpRecipe_0.Error) DO
		MpRecipe_0();
	END_WHILE
	Parameters := ParametersPreview;

	HmiRecipe.Parameters.LastLoadedProductRecipe := MpRecipe_0.Info.LastLoadedRecipe;
	HmiRecipe.Parameters.LastLoadedConfigRecipe := MACHINE_FILENAME;
	MpRecipe_0.ErrorReset := MpRecipe_0.Error;
	MpRecipe_0.Load := FALSE;
	MpRecipe_0();

    // Trigger update notification so that the initial parameters are copied to the process
    // might not be necessary.*****
	MpRecipe_0.UpdateNotification := TRUE;

	// Init Filemanager for exporting/importing files
	MpFileManagerUI_0.Enable := TRUE;
	MpFileManagerUI_0.MpLink := ADR(gMpLinkFileManagerUIRecipe);
	MpFileManagerUI_0.UIConnect := ADR(MpFileManagerUIConnect);
	MpFileManagerUI_0.UISetup.FileListSize := SIZEOF(MpFileManagerUIConnect.File.List.Items) / SIZEOF(MpFileManagerUIConnect.File.List.Items[0]);
	MpFileManagerUIConnect.DeviceList.DeviceNames[0] := 'mappRecipeFiles';
	MpFileManagerUIConnect.DeviceList.DeviceNames[1] := '';
	MpFileManagerUI_0();

	HmiRecipe.Status.HMIcommand := REC_HMI_WAIT;

END_PROGRAM

PROGRAM _CYCLIC

	// Call actions
	FormatDeviceDataProvider;
	LoadPreview;
	RecipeHMIcommands;
	FileCopyOperation;

    // Reset category after saving is done, category should be reset so that autosave files contain ALL the parameters
    IF EDGEPOS(MpRecipeUIConnect.Status = mpRECIPE_UI_STATUS_IDLE) AND ((NOT MpRecipeUIConnect.Recipe.Load) AND (NOT MpRecipeUIConnect.Recipe.Save)) THEN
        // Check if 'Product' category has been loaded
        IF ((brsstrcmp(ADR(HmiRecipe.Parameters.Category), ADR(PRODUCT_CATEGORY)) = 0) AND (HmiRecipe.Parameters.LastStatus = mpRECIPE_UI_STATUS_LOAD)) THEN
			HmiRecipe.Parameters.LastLoadedProductRecipe := MpRecipe_0.Info.LastLoadedRecipe;
			MpRecipe_0.UpdateNotification := TRUE;
		ELSIF ((brsstrcmp(ADR(HmiRecipe.Parameters.Category), ADR(MACHINE_CATEGORY)) = 0) AND (HmiRecipe.Parameters.LastStatus = mpRECIPE_UI_STATUS_LOAD)) THEN
			HmiRecipe.Parameters.LastLoadedConfigRecipe := MpRecipe_0.Info.LastLoadedRecipe;
			MpRecipe_0.UpdateNotification := TRUE;
        END_IF
		// Trigger a reload of the preview parameters
        HmiRecipe.Parameters.LastSelectedIndex := HmiRecipe.Parameters.LastSelectedIndex + 1;
        brsstrcpy(ADR(HmiRecipe.Parameters.Category), ADR(PRODUCT_CATEGORY));
    END_IF
    HmiRecipe.Parameters.LastStatus := MpRecipeUIConnect.Status;
	HmiRecipe.Parameters.ActiveRecipe := MpRecipeUIConnect.Recipe.List.Names[MpRecipeUIConnect.Recipe.List.SelectedIndex];

    // Save current recipe
    IF (HmiRecipe.Commands.SaveCurrentRecipe = TRUE) AND NOT (MpRecipe_0.Load OR MpRecipe_0.Save OR MpRecipe_0.UpdateNotification) THEN
		HmiRecipe.Parameters.FileName := HmiRecipe.Parameters.LastLoadedProductRecipe;
        DTGetTime_0(enable := TRUE);
        Header.DateTime := DTGetTime_0.DT1;
        Header.Name := HmiRecipe.Parameters.FileName;
        Header.Description := '';
        MpRecipe_0.Save := TRUE;
        HmiRecipe.Commands.SaveCurrentRecipe := FALSE;
    END_IF

	// Reset commands on MpRecipe FUB
	IF MpRecipe_0.CommandDone THEN
		// Set update notification for machine category
		IF ((brsstrcmp(ADR(HmiRecipe.Parameters.Category), ADR(MACHINE_CATEGORY)) = 0) AND (MpRecipe_0.Save = TRUE)) THEN
			MpRecipe_0.UpdateNotification := TRUE;
			MpRecipe_0.Load := FALSE;
			MpRecipe_0.Save := FALSE;
		ELSE
			MpRecipe_0.UpdateNotification := FALSE;
			MpRecipe_0.Load := FALSE;
			MpRecipe_0.Save := FALSE;
			HmiRecipe.Parameters.Category := PRODUCT_CATEGORY;
			HmiRecipe.Parameters.FileName := 'Default.par';
        END_IF
    END_IF

	// Error reset
	IF NOT MpRecipe_0.Error THEN
		MpRecipe_0.ErrorReset := FALSE;
	END_IF

	IF NOT MpRecipeUI_0.Error THEN
		MpRecipeUI_0.ErrorReset := FALSE;
	END_IF

	// Assign MpLinks
	MpRecipe_0.MpLink := ADR(gMpLinkRecipeXml);
	MpRecipeUI_0.MpLink := ADR(gMpLinkRecipeXml);
	MpFileManagerUI_0.MpLink := ADR(gMpLinkFileManagerUIRecipe);
	MpRecipeRegPar_PreviewPar.MpLink := ADR(gMpLinkRecipeXml);
	MpRecipeRegPar_PreviewCfg.MpLink := ADR(gMpLinkRecipeXml);

	// Call function blocks
	MpRecipe_0();
	MpRecipeUI_0();
	MpFileManagerUI_0();
	MpRecipeRegPar_PreviewPar();
	MpRecipeRegPar_PreviewCfg();

END_PROGRAM

PROGRAM _EXIT

	// Disable the function blocls to unlink the MpLinks
	MpRecipe_0.Enable := FALSE;
	MpRecipeUI_0.Enable := FALSE;
	MpRecipeRegPar_PreviewPar.Enable := FALSE;
	MpRecipeRegPar_PreviewCfg.Enable := FALSE;
	MpFileManagerUI_0.Enable := FALSE;

	// Call function blocks
	MpRecipe_0();
	MpRecipeUI_0();
	MpRecipeRegPar_PreviewPar();
	MpRecipeRegPar_PreviewCfg();
	MpFileManagerUI_0();

END_PROGRAM
```
